// TIA Portal project "IPC200_V15" (V15)

(* hardware
DEVICE "Estación SIMATIC 1200_1"  S71200.Device
   slot 0: "Rack S7-1200"  Rack  V1.0
   slot 1: "IPC201C"  CPU 1214C DC/DC/DC  6ES7 214-1AG40-0XB0  V4.0
   slot 2: "DI8 x 24V DC / DQ8 x relé_1"  6ES7 223-1BH32-0XB0  V2.0
   slot 3: "AI4 x 13bits_1"  6ES7 231-4HD32-0XB0  V2.0
   slot 4: "AQ4 x 14 bits_1"  6ES7 232-4HD32-0XB0  V2.0
DEVICE "S7-1200 station_1"  S7-1200 Station
   slot 0: "Rack_0"  Rack  V1.0
   slot 1: "IPC202B"  CPU 1214C DC/DC/DC  6ES7 214-1AG40-0XB0  V4.0
   slot 2: "DI 16x24VDC_1"  6ES7 221-1BH32-0XB0  V2.0
   slot 3: "DQ 8x24VDC _1"  6ES7 222-1BF32-0XB0  V2.0
DEVICE "S7-1200 station_2"  S7-1200 Station
   slot 0: "Rack_0"  S7-1200 Rack  Rack  V1.0
   slot 1: "PLC_1"  CPU 1214C DC/DC/DC  6ES7 214-1AG40-0XB0  V4.2
   slot 2: "DI 8/DQ 8x24VDC_1"  6ES7 223-1BH32-0XB0  V2.0
   slot 3: "AI 4x13BIT_1"  6ES7 231-4HD32-0XB0  V2.0
   slot 4: "AI 4x13BIT_2"  6ES7 231-4HD32-0XB0  V2.0
*)

// ===== PLC "IPC201C"  CPU 1214C DC/DC/DC =====

VAR_GLOBAL   // PLC tag table "Tabla de variables estándar"
   "A4+" AT %Q0.0 : Bool;   // Auxiliar tank output valve
   "A1+" AT %Q0.1 : Bool;   // Left tank output valve
   "B1+" AT %Q0.2 : Bool;   // Left tank input valve
   "A2+" AT %Q0.3 : Bool;   // Central tank output valve
   "B2+" AT %Q0.4 : Bool;   // Central tank input valve
   "P3+" AT %Q0.5 : Bool;   // Right tank pressure input valve
   "B3+" AT %Q0.6 : Bool;   // Right tank input valve
   "BR" AT %Q0.7 : Bool;   // Red light
   "Invert_VBus" AT %Q1.0 : Bool;   // Switch polarity Peltier cells and run fan
   "plc_reg" AT %Q1.1 : Bool;   // Switch analogue inputs to PLC
   "plc_reg0" AT %Q2.0 : Bool;   // Proportional valve control value from PLC
   "start" AT %I0.0 : Bool;   // Start pushbutton
   "stop" AT %I0.1 : Bool;   // Stop pushbutton
   "I_II" AT %I0.2 : Bool;   // Regulator/PLC
   "reset" AT %I0.3 : Bool;   // Reset pushbutton
   "max1" AT %I0.4 : Bool;   // Maximum left tank level
   "min1" AT %I0.5 : Bool;   // Minimum left tank level
   "max2" AT %I0.6 : Bool;   // Maximum central tank level
   "min2" AT %I0.7 : Bool;   // Minimum central tank level
   "max3" AT %I1.0 : Bool;   // Maximum right tank level
   "min3" AT %I1.1 : Bool;   // Minimum right tank level
   "ps3_out1" AT %I1.2 : Bool;   // Right tank pressure output 1
   "ps3_out2" AT %I1.3 : Bool;   // Right tank pressure output 2
   "dis1_out1" AT %I1.4 : Bool;   // Central tank level output 1
   "dis1_out2" AT %I1.5 : Bool;   // Central tank level output 2
   "dis2_out1" AT %I2.0 : Bool;   // Flow output 1
   "dis2_out2" AT %I2.1 : Bool;   // Flow output 2
   "AnOut1_ITV" AT %MW10 : Int;
   "AnOut2_PV" AT %MW12 : Int;
   "AnOut3_CP" AT %MW14 : Int;
   "AnOut4_PUMP" AT %MW16 : Int;
   "VP_Temp" AT %MW30 : Int;
   "VP_Flow" AT %MW32 : Int;
   "VP_Level" AT %MW34 : Int;
   "VP_P1" AT %MW36 : Int;
   "PID_in_SP" AT %MW88 : Int;
   "PID_out_CS" AT %MW90 : Int;
   "VP_Temp_real" AT %MD40 : Real;
   "VP_Flow_real" AT %MD44 : Real;
   "VP_Level_real" AT %MD48 : Real;
   "VP_Pressure_DEP1_real" AT %MD52 : Real;
   "VP_Pressure_DEP3_real" AT %MD56 : Real;
   "PID_out_CS_real" AT %MD76 : Real;
   "PID_out_Error_real" AT %MD80 : Real;
   "PID_in_SP_real" AT %MD84 : Real;
   "PID_in_PV_real" AT %MD92 : Real;
   "PID_EN" AT %M1.0 : Bool;
   "TK1_MIN" AT %M1.1 : Bool;   // Minimum level reached in DEP1
   "TK2_MIN" AT %M1.2 : Bool;   // Minimum level reached in DEP2
   "TK3_MIN" AT %M1.3 : Bool;   // Minimum level reached in DEP3
   "Running" AT %M1.4 : Bool;   // Station running
   "Set_P" AT %M1.5 : Bool;
   "Set_I" AT %M1.6 : Bool;
   "Set_D" AT %M1.7 : Bool;
   "Run_PID" AT %M2.0 : Bool;   // Activation instruction of PID
   "ITV_out" AT %QW144 : Word;   // Analogue output of ITV
   "P3_out" AT %QW146 : Word;   // Analogue output of proportional valve
   "CP_out" AT %QW148 : Word;   // Analogue output of Peltier cells
   "PUMP_out" AT %QW150 : Word;   // Analogue output of pump
   "FLOW_in" AT %IW114 : Word;   // Value of flow
   "LEVEL_in" AT %IW116 : Word;   // Value of level
   "ITV_in" AT %IW64 : Word;   // Value of pressure in left tank (ITV)
   "P3_in" AT %IW118 : Word;   // Value of pressure in right tank
   "VP_P3" AT %MW38 : Int;
   "TEMP_in" AT %IW112 : Word;   // Value of temperature
   "All_off" AT %M2.7 : Bool;
   "Step_0" AT %M3.0 : Bool;   // Step_0 - Waiting for the station 2 signal
   "Step_1" AT %M3.1 : Bool;   // Step_1 - Start to fill the can
   "Step_2" AT %M3.2 : Bool;   // Step_2 - Stop to fill the can
   "Peltier_V_scada" AT %M20.0 : Bool;   // PC-->PLC
   "Motor_scada" AT %M20.5 : Bool;   // PC-->PLC
   "Fan_scada" AT %M20.6 : Bool;   // PC-->PLC
   "A1+_scada" AT %M21.0 : Bool;   // PC-->PLC
   "B1+_scada" AT %M21.1 : Bool;   // PC-->PLC
   "A2+_scada" AT %M21.2 : Bool;   // PC-->PLC
   "B2+_scada" AT %M21.3 : Bool;   // PC-->PLC
   "P3+_scada" AT %M21.4 : Bool;   // PC-->PLC
   "B3+_scada" AT %M21.5 : Bool;   // PC-->PLC
   "A4+_scada" AT %M21.6 : Bool;   // PC-->PLC
   "A5+_scada" AT %M21.7 : Bool;   // PC-->PLC
   "P_Temp1" AT %M23.0 : Bool;   // PC-->PLC
   "PID_Reverse" AT %M23.1 : Bool;   // PC-->PLC // Reversal of working mode for the cooling action
   "P_Level1" AT %M23.2 : Bool;   // PC-->PLC
   "P_Level2" AT %M23.3 : Bool;   // PC-->PLC
   "P_Level3" AT %M23.4 : Bool;   // PC-->PLC
   "P_Flow1" AT %M23.5 : Bool;   // PC-->PLC
   "P_Flow2" AT %M23.6 : Bool;   // PC-->PLC
   "P_Flow3" AT %M23.7 : Bool;   // PC-->PLC
   "B1+_show_scada" AT %M24.0 : Bool;   // PLC-->PC
   "A2+_show_scada" AT %M24.1 : Bool;   // PLC-->PC
   "B2+_show_scada" AT %M24.2 : Bool;   // PLC-->PC
   "P3+_show_scada" AT %M24.3 : Bool;   // PLC-->PC
   "B3+_show_scada" AT %M24.4 : Bool;   // PLC-->PC
   "A4+_show_scada" AT %M24.5 : Bool;   // PLC-->PC
   "A5+_show_scada" AT %M24.6 : Bool;   // PLC-->PC
   "Min1_scada" AT %M25.0 : Bool;   // PLC-->PC
   "Min2_scada" AT %M25.1 : Bool;   // PLC-->PC
   "Min3_scada" AT %M25.2 : Bool;   // PLC-->PC
   "Max1_scada" AT %M25.3 : Bool;   // PLC-->PC
   "Max2_scada" AT %M25.4 : Bool;   // PLC-->PC
   "Max3_scada" AT %M25.5 : Bool;   // PLC-->PC
   "I_II_scada" AT %M25.6 : Bool;   // PLC-->PC
   "A1+_show_scada" AT %M25.7 : Bool;   // PLC-->PC
   "start_scada" AT %M29.6 : Bool;   // Start from the SCADA
   "stop_scada" AT %M29.7 : Bool;   // Stop from the SCADA
   "Tag_11" AT %MW20 : Word;
   "Clock_Byte" AT %MB0 : Byte;
   "Clock_10Hz" AT %M0.0 : Bool;
   "Clock_5Hz" AT %M0.1 : Bool;
   "Clock_2.5Hz" AT %M0.2 : Bool;
   "Clock_2Hz" AT %M0.3 : Bool;
   "Clock_1.25Hz" AT %M0.4 : Bool;
   "Clock_1Hz" AT %M0.5 : Bool;
   "Clock_0.625Hz" AT %M0.6 : Bool;
   "Clock_0.5Hz" AT %M0.7 : Bool;
   "P_Gain_scada_real" AT %MD60 : Real;
   "I_Time_scada_real" AT %MD64 : Real;
   "D_Time_scada_real" AT %MD68 : Real;
   "plc_reg1" AT %Q2.1 : Bool;   // ITV SetPoint from PLC
   "event_flow" AT %Q2.2 : Bool;   // Stop industrial flow controller
   "Temp1_E5CNH" AT %M22.0 : Bool;   // PC-->PLC
   "Level_aux1" AT %MD72 : UDInt;
   "Level_aux2" AT %MD96 : UDInt;
   "Level_aux3" AT %MW100 : Int;
   "Tag_10" AT %MW22 : Word;
   "Temp2_E5CNH" AT %M22.1 : Bool;   // PC-->PLC
   "Tag_13" AT %M589.0 : Bool;
   "P_Gain" AT %MD102 : Real;
   "I_Time" AT %MD106 : Real;
   "D_Time" AT %MD110 : Real;
   "P_Gain_scada" AT %MD114 : DWord;
   "I_Time_scada" AT %MD118 : DWord;
   "D_Time_scada" AT %MD122 : DWord;
   "Tag_14" AT %M400.0 : Bool;
   "Tag_15" AT %M589.1 : Bool;
   "Tag_16" AT %M589.2 : Bool;
   "VP_Temp_aux" AT %MW126 : Int;
   "PID_in_SP_aux" AT %MW128 : Int;
   "event_level" AT %Q2.3 : Bool;   // Stop industrial level controller
   "plc_reg2" AT %Q2.4 : Bool;   // Switch between flow and level control
   "A5+" AT %Q2.5 : Bool;   // Pump run
   "PLC_reg_sensor_scada" AT %M20.1 : Bool;   // PC-->PLC
   "PLC_reg0_scada" AT %M20.2 : Bool;   // PC-->PLC
   "PLC_reg1_scada" AT %M20.3 : Bool;   // PC-->PLC
   "PLC_reg2_scada" AT %M20.4 : Bool;   // PC-->PLC
   "Level1_E5CNH" AT %M22.2 : Bool;   // PC-->PLC
   "Level2_E5CNH" AT %M22.3 : Bool;   // PC-->PLC
   "Level3_E5CNH" AT %M22.4 : Bool;   // PC-->PLC
   "Flow1_E5CNH" AT %M22.5 : Bool;   // PC-->PLC
   "Flow2_E5CNH" AT %M22.6 : Bool;   // PC-->PLC
   "Flow3_E5CNH" AT %M22.7 : Bool;   // PC-->PLC
   "IPC2_on" AT %I10.0 : Bool;   // IPC202 active
   "IPC1_StartCycle" AT %I10.1 : Bool;   // Start cycle in IPC201C from IPC202
   "IPC1_on" AT %Q10.0 : Bool;   // IPC201C active to IPC202
   "IPC1_end" AT %Q10.1 : Bool;   // End cycle of IPC201C to IPC202
   "IPC1_full" AT %Q10.2 : Bool;   // Central tank full in IPC201C to IPC202
   "Tag_1" AT %IB10 : Byte;
   "TEMP_PRG" AT %M11.0 : Bool;   // Temporary parameter
   "PRG_FLAG" AT %M11.3 : Bool;   // Program is running
   "KORAK" AT %MW110 : UInt;
END_VAR

DATA_BLOCK "apple_juice_program_DB"   // DB45
{ S7_Optimized_Access := 'TRUE' }
VERSION : 0.1
// stored: InstanceOfName APPLE_JUICE_PROCESS
"APPLE_JUICE_PROCESS"
BEGIN
END_DATA_BLOCK

// folder: System blocks/Program resources

DATA_BLOCK "TIMER_1"   // DB5
{ S7_Optimized_Access := 'TRUE' }
AUTHOR : Simatic
FAMILY : IEC
NAME : IEC_TMR
VERSION : 1.0
// stored: InstanceOfName IEC_TIMER
"IEC_TIMER"
BEGIN
END_DATA_BLOCK

DATA_BLOCK "TIMER_2"   // DB6
{ S7_Optimized_Access := 'TRUE' }
AUTHOR : Simatic
FAMILY : IEC
NAME : IEC_TMR
VERSION : 1.0
// stored: InstanceOfName IEC_TIMER
"IEC_TIMER"
BEGIN
END_DATA_BLOCK

DATA_BLOCK "TIMER_3"   // DB7
{ S7_Optimized_Access := 'TRUE' }
AUTHOR : Simatic
FAMILY : IEC
NAME : IEC_TMR
VERSION : 1.0
// stored: InstanceOfName IEC_TIMER
"IEC_TIMER"
BEGIN
END_DATA_BLOCK

DATA_BLOCK "TIMER_4"   // DB8
{ S7_Optimized_Access := 'TRUE' }
AUTHOR : Simatic
FAMILY : IEC
NAME : IEC_TMR
VERSION : 1.0
// stored: InstanceOfName IEC_TIMER
"IEC_TIMER"
BEGIN
END_DATA_BLOCK

DATA_BLOCK "TIMER_5"   // DB9
{ S7_Optimized_Access := 'TRUE' }
AUTHOR : Simatic
FAMILY : IEC
NAME : IEC_TMR
VERSION : 1.0
// stored: InstanceOfName IEC_TIMER
"IEC_TIMER"
BEGIN
END_DATA_BLOCK

DATA_BLOCK "TIMER_6"   // DB10
{ S7_Optimized_Access := 'TRUE' }
AUTHOR : Simatic
FAMILY : IEC
NAME : IEC_TMR
VERSION : 1.0
// stored: InstanceOfName IEC_TIMER
"IEC_TIMER"
BEGIN
END_DATA_BLOCK

DATA_BLOCK "TIMER_7"   // DB11
{ S7_Optimized_Access := 'TRUE' }
AUTHOR : Simatic
FAMILY : IEC
NAME : IEC_TMR
VERSION : 1.0
// stored: InstanceOfName IEC_TIMER
"IEC_TIMER"
BEGIN
END_DATA_BLOCK

DATA_BLOCK "TIMER_8"   // DB12
{ S7_Optimized_Access := 'TRUE' }
AUTHOR : Simatic
FAMILY : IEC
NAME : IEC_TMR
VERSION : 1.0
// stored: InstanceOfName IEC_TIMER
"IEC_TIMER"
BEGIN
END_DATA_BLOCK

DATA_BLOCK "TIMER_9"   // DB13
{ S7_Optimized_Access := 'TRUE' }
AUTHOR : Simatic
FAMILY : IEC
NAME : IEC_TMR
VERSION : 1.0
// stored: InstanceOfName IEC_TIMER
"IEC_TIMER"
BEGIN
END_DATA_BLOCK

DATA_BLOCK "TIMER_PROG_2"   // DB17
{ S7_Optimized_Access := 'TRUE' }
AUTHOR : Simatic
FAMILY : IEC
NAME : IEC_TMR
VERSION : 1.0
// stored: InstanceOfName IEC_TIMER
"IEC_TIMER"
BEGIN
END_DATA_BLOCK

DATA_BLOCK "TIMER_PROG_1"   // DB19
{ S7_Optimized_Access := 'TRUE' }
AUTHOR : Simatic
FAMILY : IEC
NAME : IEC_TMR
VERSION : 1.0
// stored: InstanceOfName IEC_TIMER
"IEC_TIMER"
BEGIN
END_DATA_BLOCK

DATA_BLOCK "TIMER_PROG_3"   // DB20
{ S7_Optimized_Access := 'TRUE' }
AUTHOR : Simatic
FAMILY : IEC
NAME : IEC_TMR
VERSION : 1.0
// stored: InstanceOfName IEC_TIMER
"IEC_TIMER"
BEGIN
END_DATA_BLOCK

DATA_BLOCK "TIMER_PROG_4"   // DB21
{ S7_Optimized_Access := 'TRUE' }
AUTHOR : Simatic
FAMILY : IEC
NAME : IEC_TMR
VERSION : 1.0
// stored: InstanceOfName IEC_TIMER
"IEC_TIMER"
BEGIN
END_DATA_BLOCK

DATA_BLOCK "TIMER_PROG_5"   // DB22
{ S7_Optimized_Access := 'TRUE' }
AUTHOR : Simatic
FAMILY : IEC
NAME : IEC_TMR
VERSION : 1.0
// stored: InstanceOfName IEC_TIMER
"IEC_TIMER"
BEGIN
END_DATA_BLOCK

DATA_BLOCK "TIMER_PROG_6"   // DB23
{ S7_Optimized_Access := 'TRUE' }
AUTHOR : Simatic
FAMILY : IEC
NAME : IEC_TMR
VERSION : 1.0
// stored: InstanceOfName IEC_TIMER
"IEC_TIMER"
BEGIN
END_DATA_BLOCK

DATA_BLOCK "TIMER_PROG_7"   // DB24
{ S7_Optimized_Access := 'TRUE' }
AUTHOR : Simatic
FAMILY : IEC
NAME : IEC_TMR
VERSION : 1.0
// stored: InstanceOfName IEC_TIMER
"IEC_TIMER"
BEGIN
END_DATA_BLOCK

DATA_BLOCK "TIMER_PROG_8"   // DB25
{ S7_Optimized_Access := 'TRUE' }
AUTHOR : Simatic
FAMILY : IEC
NAME : IEC_TMR
VERSION : 1.0
// stored: InstanceOfName IEC_TIMER
"IEC_TIMER"
BEGIN
END_DATA_BLOCK

DATA_BLOCK "TIMER_PROG_9"   // DB26
{ S7_Optimized_Access := 'TRUE' }
AUTHOR : Simatic
FAMILY : IEC
NAME : IEC_TMR
VERSION : 1.0
// stored: InstanceOfName IEC_TIMER
"IEC_TIMER"
BEGIN
END_DATA_BLOCK

DATA_BLOCK "TIMER_PROG_10"   // DB27
{ S7_Optimized_Access := 'TRUE' }
AUTHOR : Simatic
FAMILY : IEC
NAME : IEC_TMR
VERSION : 1.0
// stored: InstanceOfName IEC_TIMER
"IEC_TIMER"
BEGIN
END_DATA_BLOCK

DATA_BLOCK "TIMER_PROG_24"   // DB28
{ S7_Optimized_Access := 'TRUE' }
AUTHOR : Simatic
FAMILY : IEC
NAME : IEC_TMR
VERSION : 1.0
// stored: InstanceOfName IEC_TIMER
"IEC_TIMER"
BEGIN
END_DATA_BLOCK

DATA_BLOCK "TIMER_PROG_12"   // DB29
{ S7_Optimized_Access := 'TRUE' }
AUTHOR : Simatic
FAMILY : IEC
NAME : IEC_TMR
VERSION : 1.0
// stored: InstanceOfName IEC_TIMER
"IEC_TIMER"
BEGIN
END_DATA_BLOCK

DATA_BLOCK "IEC_Counter_0_DB"   // DB30
{ S7_Optimized_Access := 'TRUE' }
AUTHOR : Simatic
FAMILY : IEC
NAME : CNTR
VERSION : 1.0
// stored: InstanceOfName IEC_COUNTER
"IEC_COUNTER"
BEGIN
END_DATA_BLOCK

DATA_BLOCK "TIMER_PROG_13"   // DB31
{ S7_Optimized_Access := 'TRUE' }
AUTHOR : Simatic
FAMILY : IEC
NAME : IEC_TMR
VERSION : 1.0
// stored: InstanceOfName IEC_TIMER
"IEC_TIMER"
BEGIN
END_DATA_BLOCK

DATA_BLOCK "IEC_Counter_0_DB_1"   // DB32
{ S7_Optimized_Access := 'TRUE' }
AUTHOR : Simatic
FAMILY : IEC
NAME : CNTR
VERSION : 1.0
// stored: InstanceOfName IEC_COUNTER
"IEC_COUNTER"
BEGIN
END_DATA_BLOCK

DATA_BLOCK "TIMER_PROG_14"   // DB33
{ S7_Optimized_Access := 'TRUE' }
AUTHOR : Simatic
FAMILY : IEC
NAME : IEC_TMR
VERSION : 1.0
// stored: InstanceOfName IEC_TIMER
"IEC_TIMER"
BEGIN
END_DATA_BLOCK

DATA_BLOCK "TIMER_PROG_15"   // DB34
{ S7_Optimized_Access := 'TRUE' }
AUTHOR : Simatic
FAMILY : IEC
NAME : IEC_TMR
VERSION : 1.0
// stored: InstanceOfName IEC_TIMER
"IEC_TIMER"
BEGIN
END_DATA_BLOCK

DATA_BLOCK "TIMER_PROG_16"   // DB35
{ S7_Optimized_Access := 'TRUE' }
AUTHOR : Simatic
FAMILY : IEC
NAME : IEC_TMR
VERSION : 1.0
// stored: InstanceOfName IEC_TIMER
"IEC_TIMER"
BEGIN
END_DATA_BLOCK

DATA_BLOCK "TIMER_PROG_17"   // DB36
{ S7_Optimized_Access := 'TRUE' }
AUTHOR : Simatic
FAMILY : IEC
NAME : IEC_TMR
VERSION : 1.0
// stored: InstanceOfName IEC_TIMER
"IEC_TIMER"
BEGIN
END_DATA_BLOCK

DATA_BLOCK "TIMER_PROG_18"   // DB37
{ S7_Optimized_Access := 'TRUE' }
AUTHOR : Simatic
FAMILY : IEC
NAME : IEC_TMR
VERSION : 1.0
// stored: InstanceOfName IEC_TIMER
"IEC_TIMER"
BEGIN
END_DATA_BLOCK

DATA_BLOCK "IEC_Counter_0_DB_2"   // DB38
{ S7_Optimized_Access := 'TRUE' }
AUTHOR : Simatic
FAMILY : IEC
NAME : CNTR
VERSION : 1.0
// stored: InstanceOfName IEC_COUNTER
"IEC_COUNTER"
BEGIN
END_DATA_BLOCK

DATA_BLOCK "TIMER_PROG_19"   // DB39
{ S7_Optimized_Access := 'TRUE' }
AUTHOR : Simatic
FAMILY : IEC
NAME : IEC_TMR
VERSION : 1.0
// stored: InstanceOfName IEC_TIMER
"IEC_TIMER"
BEGIN
END_DATA_BLOCK

DATA_BLOCK "TIMER_PROG_20"   // DB40
{ S7_Optimized_Access := 'TRUE' }
AUTHOR : Simatic
FAMILY : IEC
NAME : IEC_TMR
VERSION : 1.0
// stored: InstanceOfName IEC_TIMER
"IEC_TIMER"
BEGIN
END_DATA_BLOCK

DATA_BLOCK "TIMER_PROG_21"   // DB41
{ S7_Optimized_Access := 'TRUE' }
AUTHOR : Simatic
FAMILY : IEC
NAME : IEC_TMR
VERSION : 1.0
// stored: InstanceOfName IEC_TIMER
"IEC_TIMER"
BEGIN
END_DATA_BLOCK

DATA_BLOCK "TIMER_PROG_22"   // DB42
{ S7_Optimized_Access := 'TRUE' }
AUTHOR : Simatic
FAMILY : IEC
NAME : IEC_TMR
VERSION : 1.0
// stored: InstanceOfName IEC_TIMER
"IEC_TIMER"
BEGIN
END_DATA_BLOCK

DATA_BLOCK "TIMER_PROG_23"   // DB43
{ S7_Optimized_Access := 'TRUE' }
AUTHOR : Simatic
FAMILY : IEC
NAME : IEC_TMR
VERSION : 1.0
// stored: InstanceOfName IEC_TIMER
"IEC_TIMER"
BEGIN
END_DATA_BLOCK

DATA_BLOCK "IEC_Counter_0_DB_3"   // DB44
{ S7_Optimized_Access := 'TRUE' }
AUTHOR : Simatic
FAMILY : IEC
NAME : CNTR
VERSION : 1.0
// stored: InstanceOfName IEC_COUNTER
"IEC_COUNTER"
BEGIN
END_DATA_BLOCK

DATA_BLOCK "IEC_Timer_0_DB_1"   // DB52
{ S7_Optimized_Access := 'TRUE' }
AUTHOR : Simatic
FAMILY : IEC
NAME : IEC_TMR
VERSION : 1.0
// stored: InstanceOfName IEC_TIMER
"IEC_TIMER"
BEGIN
END_DATA_BLOCK

DATA_BLOCK "IEC_Timer_0_DB"   // DB53
{ S7_Optimized_Access := 'TRUE' }
AUTHOR : Simatic
FAMILY : IEC
NAME : IEC_TMR
VERSION : 1.0
// stored: InstanceOfName IEC_TIMER
"IEC_TIMER"
BEGIN
END_DATA_BLOCK

// folder: (top level)

FUNCTION_BLOCK "APPLE_JUICE_PROCESS"   // FB1, SCL
{ S7_Optimized_Access := 'TRUE' }
VERSION : 0.1
   VAR
      currentState : Int := 0;
      "timer" : Time;
      onDelayCheck : Bool;
      fallingEgdeDedect1 : Bool;
      fallingEgdeDedect : Bool;
      risingEgdeDedect : Bool;
      processFinished : Bool;
   END_VAR
   VAR CONSTANT
      STATE_WAIT_FOR_START : Int := -1;
      STATE_START_FILL_WATER : Int;
      STATE_WAIT_FOR_FILL_WATER_TANK : Int := 1;
      FILL_WAIT : Time := T#5s;
      STATE_START_FILL_APPLE : Int := 2;
      STATE_WAIT_FILL_APPLE : Int := 3;
      STATE_START_FILL_APPLE_JUICE_WITH_WATER : Int := 4;
      STATE_WAIT_FILL_APPLE_JUICE_WITH_WATER : Int := 5;
      STATE_START_FILL_APPLE_JUICE_WITH_APPLE : Int := 6;
      STATE_WAIT_FILL_APPLE_JUICE_WITH_APPLE : Int := 7;
      STATE_START_FILL_OUT_APPLE : Int := 8;
      STATE_WAIT_FILL_OUT_APPLE : Int := 9;
      STATE_WAIT_FOR_NEXT_PROCESS : Int := 10;
      PUMP_CHARGE : Int := 8000;
      VALVE_CHARE : Int := 20000;
   END_VAR
BEGIN
   CASE #currentState OF
       #STATE_WAIT_FOR_START:
           "R_TRIG_DB_1"(CLK:="start",
                         Q=>#risingEgdeDedect);

           IF #risingEgdeDedect = TRUE THEN
               #currentState := #STATE_START_FILL_WATER;
           END_IF;

       #STATE_START_FILL_WATER:
           "START_LOAD_TANK"(feedback1 := "A4+",
                             feedback2 := "A5+",
                             feedback3 := "B1+",
                             command1 => "A4+_scada",
                             command2 => "A5+_scada",
                             command3 => "B1+_scada",
                             pumpValue := #PUMP_CHARGE,
                             pumpOutput => "AnOut4_PUMP",
                             routeReady => #processFinished);

           IF #processFinished = TRUE THEN
               #currentState := #STATE_WAIT_FOR_FILL_WATER_TANK;
           END_IF;

       #STATE_WAIT_FOR_FILL_WATER_TANK:
           "F_TRIG_DB"(CLK := "max1",
                       Q => #fallingEgdeDedect);

           IF #fallingEgdeDedect = TRUE OR "max1" = FALSE THEN
               "STOP_LOAD_TANK"(command1 => "A4+_scada",
                                command2 => "A5+_scada",
                                command3 => "B1+_scada",
                                pumpOutput => "AnOut4_PUMP");

               #currentState := #STATE_START_FILL_APPLE;
           END_IF;

       #STATE_START_FILL_APPLE:
           "START_LOAD_TANK"(feedback1 := "A4+",
                             feedback2 := "A5+",
                             feedback3 := "B3+",
                             command1 => "A4+_scada",
                             command2 => "A5+_scada",
                             command3 => "B3+_scada",
                             pumpValue := #PUMP_CHARGE,
                             pumpOutput => "AnOut4_PUMP",
                             routeReady => #processFinished);

           IF #processFinished = TRUE THEN
               #currentState := #STATE_WAIT_FILL_APPLE;
           END_IF;

       #STATE_WAIT_FILL_APPLE:
           "F_TRIG_DB_1"(CLK := "max3",
                         Q => #fallingEgdeDedect);

           IF #fallingEgdeDedect = TRUE OR "max3" = FALSE THEN
               "STOP_LOAD_TANK"(command1 => "A4+_scada",
                                command2 => "A5+_scada",
                                command3 => "B3+_scada",
                                pumpOutput => "AnOut4_PUMP");

               #currentState := #STATE_START_FILL_APPLE_JUICE_WITH_WATER;
           END_IF;

       #STATE_START_FILL_APPLE_JUICE_WITH_WATER:
           "START_LOAD_APPLE_JUICE_TANK"(feedback1 := "A1+",
                                         feedback2 := "B2+",
                                         command1 => "A1+_scada",
                                         command2 => "B2+_scada",
                                         regulatorCommand => "PLC_reg1_scada",
                                         analogValue := #VALVE_CHARE,
                                         analogOutput => "AnOut1_ITV",
                                         routeReady => #processFinished);

           IF #processFinished = TRUE THEN
               #currentState := #STATE_WAIT_FILL_APPLE_JUICE_WITH_WATER;
           END_IF;

       #STATE_WAIT_FILL_APPLE_JUICE_WITH_WATER:
           "R_TRIG_DB"(CLK := "min2",
                       Q => #risingEgdeDedect);

           IF #risingEgdeDedect = TRUE OR "min2" = TRUE THEN
               "STOP_LOAD_APPLE_JUICE_TANK"(command1 => "A1+_scada",
                                            command2 => "B2+_scada",
                                            regulatorCommand => "PLC_reg0_scada",
                                            analogOutput => "AnOut1_ITV");

               #currentState := #STATE_START_FILL_APPLE_JUICE_WITH_APPLE;
           END_IF;

       #STATE_START_FILL_APPLE_JUICE_WITH_APPLE:
           "START_LOAD_APPLE_JUICE_TANK"(feedback1 := "P3+",
                                         feedback2 := "B2+",
                                         command1 => "P3+_scada",
                                         command2 => "B2+_scada",
                                         regulatorCommand => "PLC_reg0_scada",
                                         analogValue := #VALVE_CHARE,
                                         analogOutput => "AnOut2_PV",
                                         routeReady => #processFinished);

           IF #processFinished = TRUE THEN
               #currentState := #STATE_WAIT_FILL_APPLE_JUICE_WITH_APPLE;
           END_IF;

       #STATE_WAIT_FILL_APPLE_JUICE_WITH_APPLE:
           "F_TRIG_DB_2"(CLK := "min3",
                         Q => #fallingEgdeDedect);
           "F_TRIG_DB_3"(CLK := "max2",
                         Q => #fallingEgdeDedect1);



           IF (#fallingEgdeDedect = TRUE OR "min3" = FALSE) OR
               (#fallingEgdeDedect1 = TRUE OR "max2" = FALSE) THEN
               "STOP_LOAD_APPLE_JUICE_TANK"(command1 => "P3+_scada",
                                            command2 => "B2+_scada",
                                            regulatorCommand => "PLC_reg1_scada",
                                            analogOutput => "AnOut2_PV");

               #currentState := #STATE_START_FILL_OUT_APPLE;
           END_IF;

       #STATE_START_FILL_OUT_APPLE:
           "FILL_APPLE_TO_BOTTLE"(feedback1 := "A2+",
                                  feedback2 := "A5+",
                                  command1 => "A2+_scada",
                                  command2 => "A5+_scada",
                                  analogValue := 8000,
                                  analogOutput => "AnOut4_PUMP",
                                  routeReady => #processFinished);

           IF #processFinished = TRUE THEN
               #currentState := #STATE_WAIT_FILL_OUT_APPLE;
           END_IF;

       #STATE_WAIT_FILL_OUT_APPLE:
           "IEC_Timer_0_DB".TON(IN := TRUE,
                                PT := T#40s,
                                Q => #onDelayCheck,
                                ET => #timer);


           IF #onDelayCheck = TRUE THEN
               "STOP_FILL_APPLE_TO_BOTTLE"(command1 => "A2+_scada",
                                           command2 => "A5+_scada",
                                           analogOutput => "AnOut4_PUMP");

               "IEC_Timer_0_DB".TON(IN := FALSE,
                                    PT := T#40s,
                                    Q => #onDelayCheck,
                                    ET => #timer);

               #currentState := #STATE_WAIT_FOR_START;
           END_IF;
   END_CASE;
END_FUNCTION_BLOCK

FUNCTION "TIMERS" : Void   // FC1, LAD
TITLE = TIMERS
{ S7_Optimized_Access := 'TRUE' }
VERSION : 0.1
BEGIN

REGION Network 1: TIMER 1
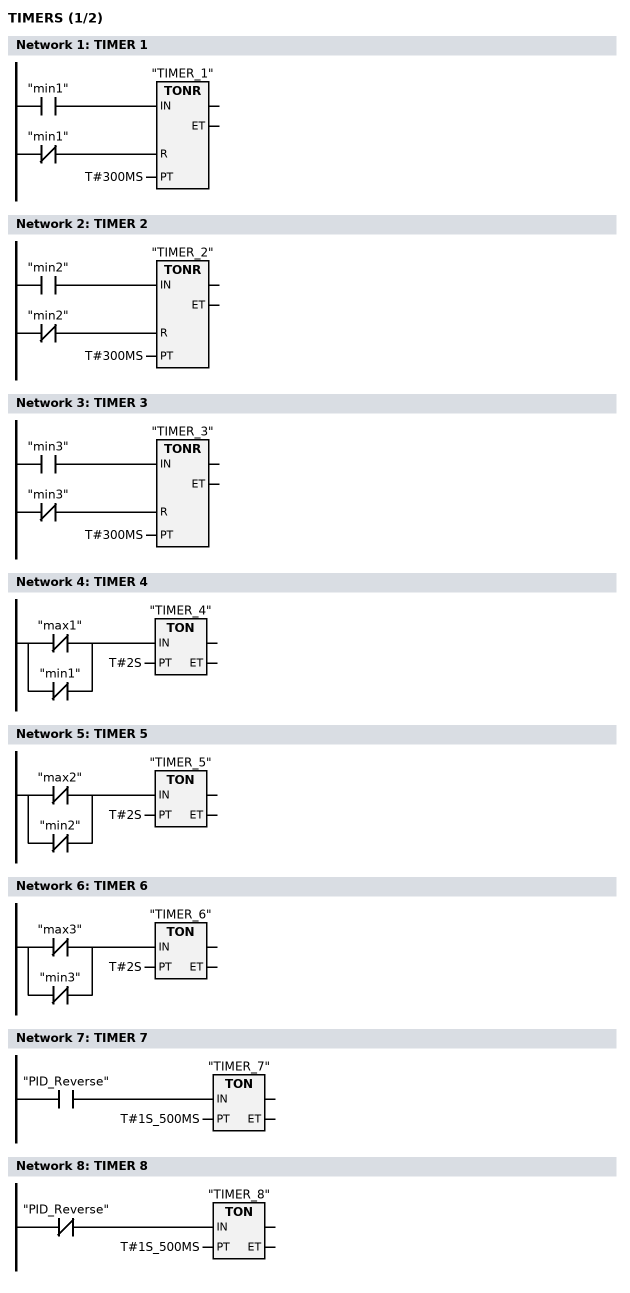
   "TIMER_1".TONR(IN := "min1", R := NOT "min1", PT := T#300MS);
END_REGION

REGION Network 2: TIMER 2
   "TIMER_2".TONR(IN := "min2", R := NOT "min2", PT := T#300MS);
END_REGION

REGION Network 3: TIMER 3
   "TIMER_3".TONR(IN := "min3", R := NOT "min3", PT := T#300MS);
END_REGION

REGION Network 4: TIMER 4
   "TIMER_4".TON(IN := NOT "max1" OR NOT "min1", PT := T#2S);
END_REGION

REGION Network 5: TIMER 5
   "TIMER_5".TON(IN := NOT "max2" OR NOT "min2", PT := T#2S);
END_REGION

REGION Network 6: TIMER 6
   "TIMER_6".TON(IN := NOT "max3" OR NOT "min3", PT := T#2S);
END_REGION

REGION Network 7: TIMER 7
   "TIMER_7".TON(IN := "PID_Reverse", PT := T#1S_500MS);
END_REGION

REGION Network 8: TIMER 8
   "TIMER_8".TON(IN := NOT "PID_Reverse", PT := T#1S_500MS);
END_REGION

REGION Network 9: TIMER 9
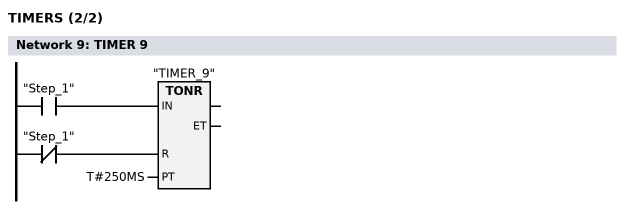
   "TIMER_9".TONR(IN := "Step_1", R := NOT "Step_1", PT := T#250MS);
END_REGION
END_FUNCTION

FUNCTION "WORKBITS" : Void   // FC2, LAD
TITLE = WORKBITS
{ S7_Optimized_Access := 'TRUE' }
VERSION : 0.1
BEGIN

REGION Network 1: TK1_MIN
   // Min level reached in DEP1
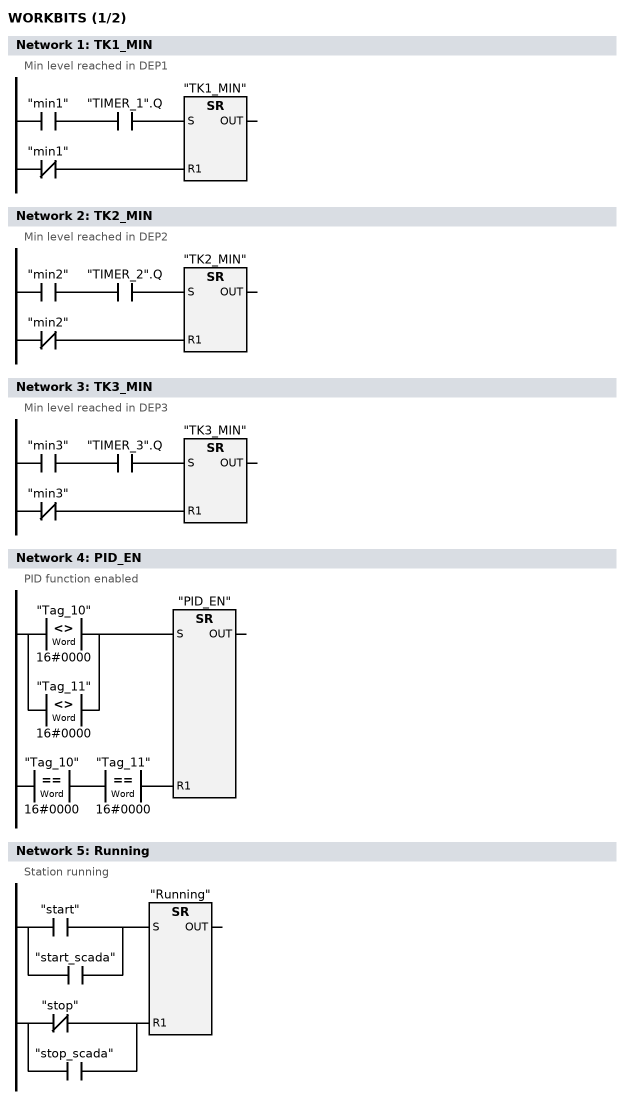
   RUNG wire#powerrail
      Contact( "min1" )
      Contact( "TIMER_1".Q )
      S_SR(operand := "TK1_MIN", r1 := wire#w1)
   END_RUNG
   RUNG wire#powerrail
      I_Contact( "min1" )
   END_RUNG wire#w1
   // the same network as SCL:
   IF "min1" AND "TIMER_1".Q THEN
       "TK1_MIN" := TRUE;   // SR flip-flop
   END_IF;
   IF NOT "min1" THEN "TK1_MIN" := FALSE; END_IF;
END_REGION

REGION Network 2: TK2_MIN
   // Min level reached in DEP2
   RUNG wire#powerrail
      Contact( "min2" )
      Contact( "TIMER_2".Q )
      S_SR(operand := "TK2_MIN", r1 := wire#w1)
   END_RUNG
   RUNG wire#powerrail
      I_Contact( "min2" )
   END_RUNG wire#w1
   // the same network as SCL:
   IF "min2" AND "TIMER_2".Q THEN
       "TK2_MIN" := TRUE;   // SR flip-flop
   END_IF;
   IF NOT "min2" THEN "TK2_MIN" := FALSE; END_IF;
END_REGION

REGION Network 3: TK3_MIN
   // Min level reached in DEP3
   RUNG wire#powerrail
      Contact( "min3" )
      Contact( "TIMER_3".Q )
      S_SR(operand := "TK3_MIN", r1 := wire#w1)
   END_RUNG
   RUNG wire#powerrail
      I_Contact( "min3" )
   END_RUNG wire#w1
   // the same network as SCL:
   IF "min3" AND "TIMER_3".Q THEN
       "TK3_MIN" := TRUE;   // SR flip-flop
   END_IF;
   IF NOT "min3" THEN "TK3_MIN" := FALSE; END_IF;
END_REGION

REGION Network 4: PID_EN
   // PID function enabled
   RUNG wire#powerrail
      { S7_Templates := "SrcType := Word" } NE_Contact(in1 := "Tag_10", in2 := 16#0000)
      wire#w1
      S_SR(operand := "PID_EN", r1 := wire#w2)
   END_RUNG
   RUNG wire#powerrail
      { S7_Templates := "SrcType := Word" } NE_Contact(in1 := "Tag_11", in2 := 16#0000)
   END_RUNG wire#w1
   RUNG wire#powerrail
      { S7_Templates := "SrcType := Word" } EQ_Contact(in1 := "Tag_10", in2 := 16#0000)
      { S7_Templates := "SrcType := Word" } EQ_Contact(in1 := "Tag_11", in2 := 16#0000)
   END_RUNG wire#w2
   // the same network as SCL:
   IF ("Tag_10" <> 16#0000) OR ("Tag_11" <> 16#0000) THEN
       "PID_EN" := TRUE;   // SR flip-flop
   END_IF;
   IF ("Tag_10" = 16#0000) AND ("Tag_11" = 16#0000) THEN "PID_EN" := FALSE; END_IF;
END_REGION

REGION Network 5: Running
   // Station running
   RUNG wire#powerrail
      Contact( "start" )
      wire#w1
      S_SR(operand := "Running", r1 := wire#w2)
   END_RUNG
   RUNG wire#powerrail
      Contact( "start_scada" )
   END_RUNG wire#w1
   RUNG wire#powerrail
      I_Contact( "stop" )
   END_RUNG wire#w2
   RUNG wire#powerrail
      Contact( "stop_scada" )
   END_RUNG wire#w2
   // the same network as SCL:
   IF "start" OR "start_scada" THEN
       "Running" := TRUE;   // SR flip-flop
   END_IF;
   IF NOT "stop" OR "stop_scada" THEN "Running" := FALSE; END_IF;
END_REGION

REGION Network 6: Run_PID
   // Activation instruction of PID
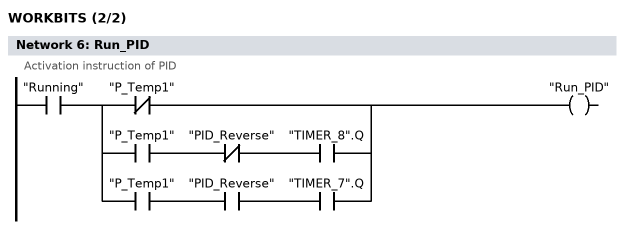
   RUNG wire#powerrail
      Contact( "Running" )
      wire#w1
      I_Contact( "P_Temp1" )
      wire#w2
      Coil( "Run_PID" )
   END_RUNG
   RUNG wire#w1
      Contact( "P_Temp1" )
      I_Contact( "PID_Reverse" )
      Contact( "TIMER_8".Q )
   END_RUNG wire#w2
   RUNG wire#w1
      Contact( "P_Temp1" )
      Contact( "PID_Reverse" )
      Contact( "TIMER_7".Q )
   END_RUNG wire#w2
   // the same network as SCL:
   "Run_PID" := "Running" AND (NOT "P_Temp1" OR ("P_Temp1" AND NOT "PID_Reverse" AND "TIMER_8".Q) OR ("P_Temp1" AND "PID_Reverse" AND "TIMER_7".Q));
END_REGION
END_FUNCTION

FUNCTION "SCADA" : Void   // FC3, LAD
TITLE = Communication between SCADA (PC) and PLC
{ S7_Optimized_Access := 'TRUE' }
VERSION : 0.1
BEGIN

REGION Network 1: PLC-->PLC
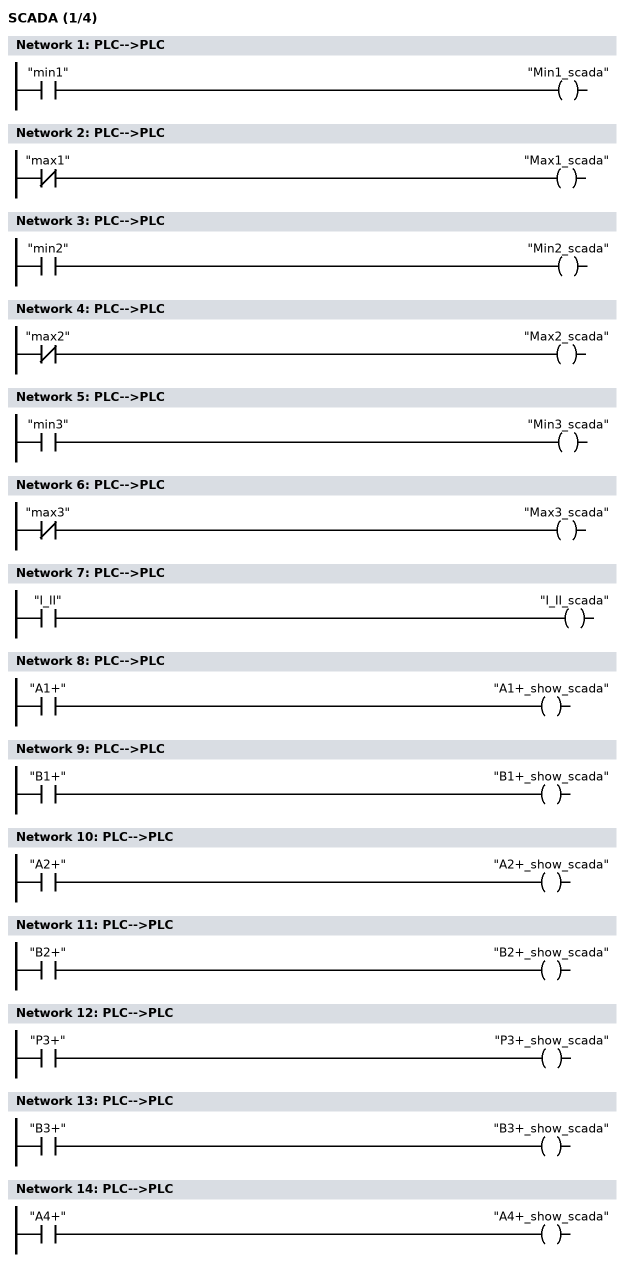
   RUNG wire#powerrail
      Contact( "min1" )
      Coil( "Min1_scada" )
   END_RUNG
   // the same network as SCL:
   "Min1_scada" := "min1";
END_REGION

REGION Network 2: PLC-->PLC
   RUNG wire#powerrail
      I_Contact( "max1" )
      Coil( "Max1_scada" )
   END_RUNG
   // the same network as SCL:
   "Max1_scada" := NOT "max1";
END_REGION

REGION Network 3: PLC-->PLC
   RUNG wire#powerrail
      Contact( "min2" )
      Coil( "Min2_scada" )
   END_RUNG
   // the same network as SCL:
   "Min2_scada" := "min2";
END_REGION

REGION Network 4: PLC-->PLC
   RUNG wire#powerrail
      I_Contact( "max2" )
      Coil( "Max2_scada" )
   END_RUNG
   // the same network as SCL:
   "Max2_scada" := NOT "max2";
END_REGION

REGION Network 5: PLC-->PLC
   RUNG wire#powerrail
      Contact( "min3" )
      Coil( "Min3_scada" )
   END_RUNG
   // the same network as SCL:
   "Min3_scada" := "min3";
END_REGION

REGION Network 6: PLC-->PLC
   RUNG wire#powerrail
      I_Contact( "max3" )
      Coil( "Max3_scada" )
   END_RUNG
   // the same network as SCL:
   "Max3_scada" := NOT "max3";
END_REGION

REGION Network 7: PLC-->PLC
   RUNG wire#powerrail
      Contact( "I_II" )
      Coil( "I_II_scada" )
   END_RUNG
   // the same network as SCL:
   "I_II_scada" := "I_II";
END_REGION

REGION Network 8: PLC-->PLC
   RUNG wire#powerrail
      Contact( "A1+" )
      Coil( "A1+_show_scada" )
   END_RUNG
   // the same network as SCL:
   "A1+_show_scada" := "A1+";
END_REGION

REGION Network 9: PLC-->PLC
   RUNG wire#powerrail
      Contact( "B1+" )
      Coil( "B1+_show_scada" )
   END_RUNG
   // the same network as SCL:
   "B1+_show_scada" := "B1+";
END_REGION

REGION Network 10: PLC-->PLC
   RUNG wire#powerrail
      Contact( "A2+" )
      Coil( "A2+_show_scada" )
   END_RUNG
   // the same network as SCL:
   "A2+_show_scada" := "A2+";
END_REGION

REGION Network 11: PLC-->PLC
   RUNG wire#powerrail
      Contact( "B2+" )
      Coil( "B2+_show_scada" )
   END_RUNG
   // the same network as SCL:
   "B2+_show_scada" := "B2+";
END_REGION

REGION Network 12: PLC-->PLC
   RUNG wire#powerrail
      Contact( "P3+" )
      Coil( "P3+_show_scada" )
   END_RUNG
   // the same network as SCL:
   "P3+_show_scada" := "P3+";
END_REGION

REGION Network 13: PLC-->PLC
   RUNG wire#powerrail
      Contact( "B3+" )
      Coil( "B3+_show_scada" )
   END_RUNG
   // the same network as SCL:
   "B3+_show_scada" := "B3+";
END_REGION

REGION Network 14: PLC-->PLC
   RUNG wire#powerrail
      Contact( "A4+" )
      Coil( "A4+_show_scada" )
   END_RUNG
   // the same network as SCL:
   "A4+_show_scada" := "A4+";
END_REGION

REGION Network 15: PLC-->PLC
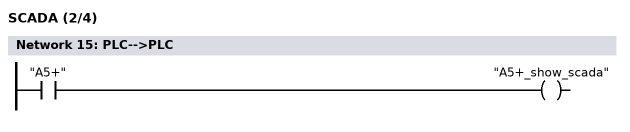
   RUNG wire#powerrail
      Contact( "A5+" )
      Coil( "A5+_show_scada" )
   END_RUNG
   // the same network as SCL:
   "A5+_show_scada" := "A5+";
END_REGION

REGION Network 16: PID PARAMETERS FROM THE SCADA
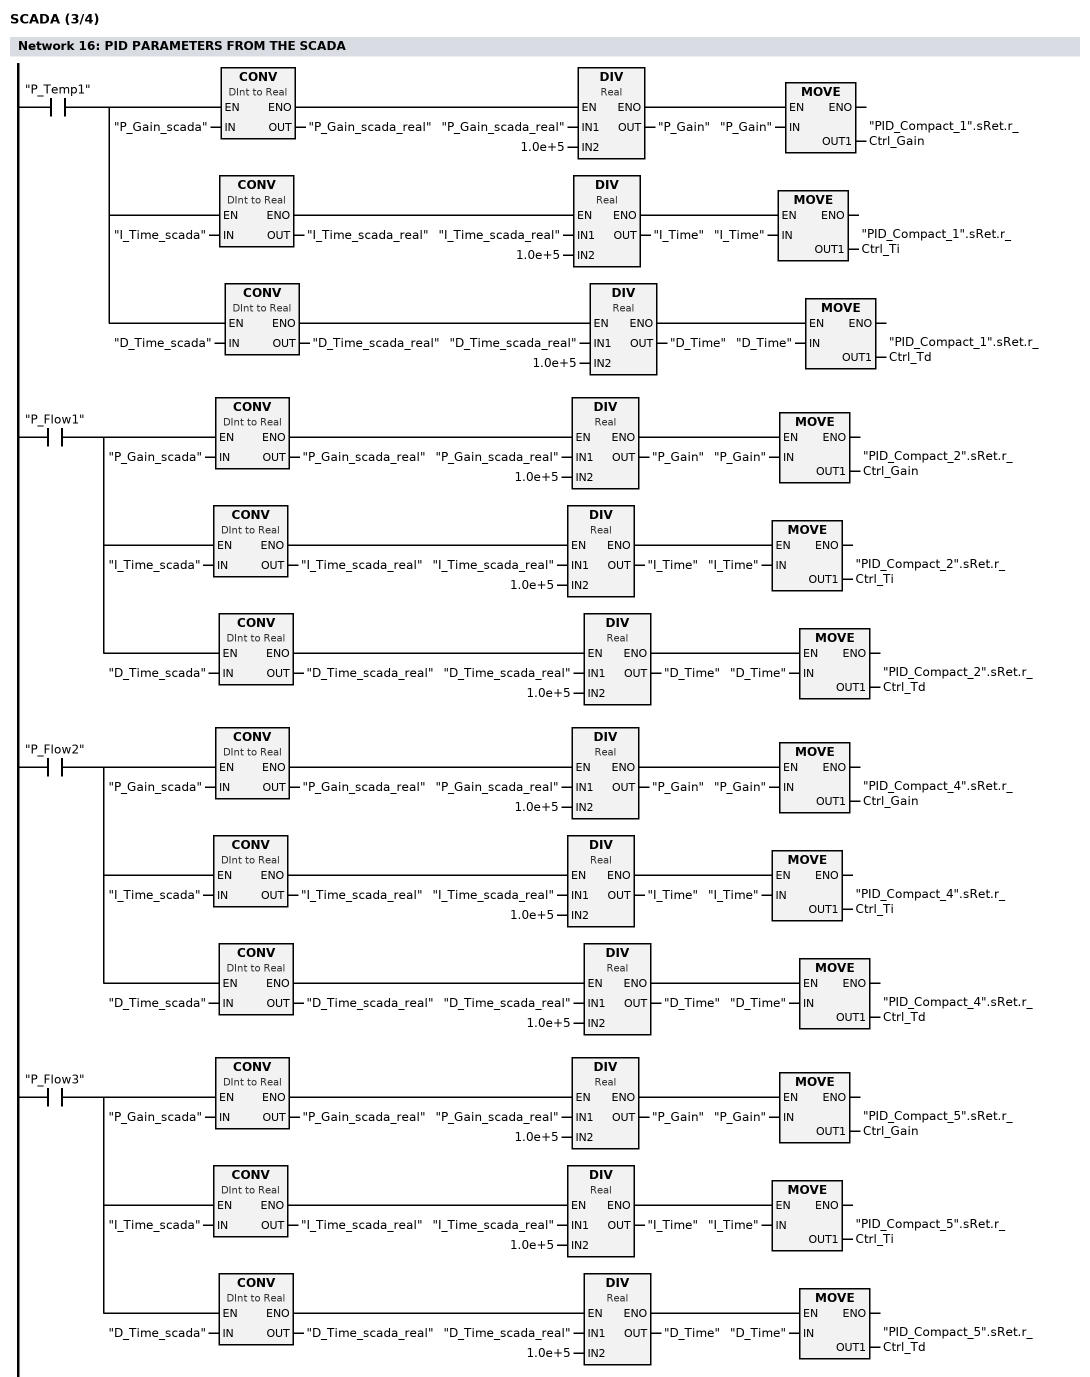
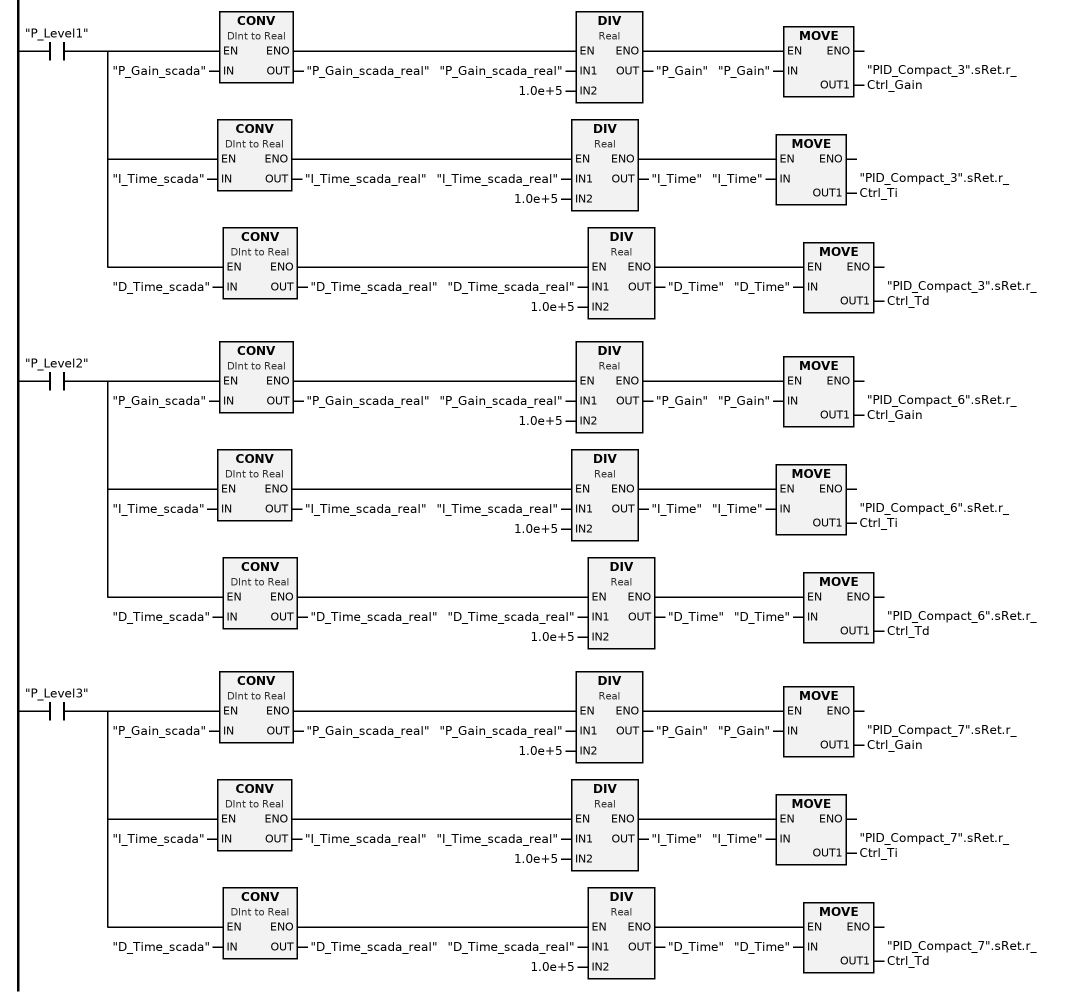
   RUNG wire#powerrail
      Contact( "P_Temp1" )
      wire#w1
      { S7_Templates := "[SrcType := DInt, DestType := Real]"; S7_GenerateENO := "TRUE" } Convert(in := "P_Gain_scada", out => "P_Gain_scada_real")
      { S7_Templates := "SrcType := Real"; S7_GenerateENO := "TRUE" } Div(in1 := "P_Gain_scada_real", in2 := 1.0e+5, out => "P_Gain")
      { S7_GenerateENO := "TRUE" } Move(in := "P_Gain", out1 => "PID_Compact_1".sRet.r_Ctrl_Gain)
   END_RUNG
   RUNG wire#w1
      { S7_Templates := "[SrcType := DInt, DestType := Real]"; S7_GenerateENO := "TRUE" } Convert(in := "I_Time_scada", out => "I_Time_scada_real")
      { S7_Templates := "SrcType := Real"; S7_GenerateENO := "TRUE" } Div(in1 := "I_Time_scada_real", in2 := 1.0e+5, out => "I_Time")
      { S7_GenerateENO := "TRUE" } Move(in := "I_Time", out1 => "PID_Compact_1".sRet.r_Ctrl_Ti)
   END_RUNG
   RUNG wire#w1
      { S7_Templates := "[SrcType := DInt, DestType := Real]"; S7_GenerateENO := "TRUE" } Convert(in := "D_Time_scada", out => "D_Time_scada_real")
      { S7_Templates := "SrcType := Real"; S7_GenerateENO := "TRUE" } Div(in1 := "D_Time_scada_real", in2 := 1.0e+5, out => "D_Time")
      { S7_GenerateENO := "TRUE" } Move(in := "D_Time", out1 => "PID_Compact_1".sRet.r_Ctrl_Td)
   END_RUNG
   RUNG wire#powerrail
      Contact( "P_Flow1" )
      wire#w2
      { S7_Templates := "[SrcType := DInt, DestType := Real]"; S7_GenerateENO := "TRUE" } Convert(in := "P_Gain_scada", out => "P_Gain_scada_real")
      { S7_Templates := "SrcType := Real"; S7_GenerateENO := "TRUE" } Div(in1 := "P_Gain_scada_real", in2 := 1.0e+5, out => "P_Gain")
      { S7_GenerateENO := "TRUE" } Move(in := "P_Gain", out1 => "PID_Compact_2".sRet.r_Ctrl_Gain)
   END_RUNG
   RUNG wire#w2
      { S7_Templates := "[SrcType := DInt, DestType := Real]"; S7_GenerateENO := "TRUE" } Convert(in := "I_Time_scada", out => "I_Time_scada_real")
      { S7_Templates := "SrcType := Real"; S7_GenerateENO := "TRUE" } Div(in1 := "I_Time_scada_real", in2 := 1.0e+5, out => "I_Time")
      { S7_GenerateENO := "TRUE" } Move(in := "I_Time", out1 => "PID_Compact_2".sRet.r_Ctrl_Ti)
   END_RUNG
   RUNG wire#w2
      { S7_Templates := "[SrcType := DInt, DestType := Real]"; S7_GenerateENO := "TRUE" } Convert(in := "D_Time_scada", out => "D_Time_scada_real")
      { S7_Templates := "SrcType := Real"; S7_GenerateENO := "TRUE" } Div(in1 := "D_Time_scada_real", in2 := 1.0e+5, out => "D_Time")
      { S7_GenerateENO := "TRUE" } Move(in := "D_Time", out1 => "PID_Compact_2".sRet.r_Ctrl_Td)
   END_RUNG
   RUNG wire#powerrail
      Contact( "P_Flow2" )
      wire#w3
      { S7_Templates := "[SrcType := DInt, DestType := Real]"; S7_GenerateENO := "TRUE" } Convert(in := "P_Gain_scada", out => "P_Gain_scada_real")
      { S7_Templates := "SrcType := Real"; S7_GenerateENO := "TRUE" } Div(in1 := "P_Gain_scada_real", in2 := 1.0e+5, out => "P_Gain")
      { S7_GenerateENO := "TRUE" } Move(in := "P_Gain", out1 => "PID_Compact_4".sRet.r_Ctrl_Gain)
   END_RUNG
   RUNG wire#w3
      { S7_Templates := "[SrcType := DInt, DestType := Real]"; S7_GenerateENO := "TRUE" } Convert(in := "I_Time_scada", out => "I_Time_scada_real")
      { S7_Templates := "SrcType := Real"; S7_GenerateENO := "TRUE" } Div(in1 := "I_Time_scada_real", in2 := 1.0e+5, out => "I_Time")
      { S7_GenerateENO := "TRUE" } Move(in := "I_Time", out1 => "PID_Compact_4".sRet.r_Ctrl_Ti)
   END_RUNG
   RUNG wire#w3
      { S7_Templates := "[SrcType := DInt, DestType := Real]"; S7_GenerateENO := "TRUE" } Convert(in := "D_Time_scada", out => "D_Time_scada_real")
      { S7_Templates := "SrcType := Real"; S7_GenerateENO := "TRUE" } Div(in1 := "D_Time_scada_real", in2 := 1.0e+5, out => "D_Time")
      { S7_GenerateENO := "TRUE" } Move(in := "D_Time", out1 => "PID_Compact_4".sRet.r_Ctrl_Td)
   END_RUNG
   RUNG wire#powerrail
      Contact( "P_Flow3" )
      wire#w4
      { S7_Templates := "[SrcType := DInt, DestType := Real]"; S7_GenerateENO := "TRUE" } Convert(in := "P_Gain_scada", out => "P_Gain_scada_real")
      { S7_Templates := "SrcType := Real"; S7_GenerateENO := "TRUE" } Div(in1 := "P_Gain_scada_real", in2 := 1.0e+5, out => "P_Gain")
      { S7_GenerateENO := "TRUE" } Move(in := "P_Gain", out1 => "PID_Compact_5".sRet.r_Ctrl_Gain)
   END_RUNG
   RUNG wire#w4
      { S7_Templates := "[SrcType := DInt, DestType := Real]"; S7_GenerateENO := "TRUE" } Convert(in := "I_Time_scada", out => "I_Time_scada_real")
      { S7_Templates := "SrcType := Real"; S7_GenerateENO := "TRUE" } Div(in1 := "I_Time_scada_real", in2 := 1.0e+5, out => "I_Time")
      { S7_GenerateENO := "TRUE" } Move(in := "I_Time", out1 => "PID_Compact_5".sRet.r_Ctrl_Ti)
   END_RUNG
   RUNG wire#w4
      { S7_Templates := "[SrcType := DInt, DestType := Real]"; S7_GenerateENO := "TRUE" } Convert(in := "D_Time_scada", out => "D_Time_scada_real")
      { S7_Templates := "SrcType := Real"; S7_GenerateENO := "TRUE" } Div(in1 := "D_Time_scada_real", in2 := 1.0e+5, out => "D_Time")
      { S7_GenerateENO := "TRUE" } Move(in := "D_Time", out1 => "PID_Compact_5".sRet.r_Ctrl_Td)
   END_RUNG
   RUNG wire#powerrail
      Contact( "P_Level1" )
      wire#w5
      { S7_Templates := "[SrcType := DInt, DestType := Real]"; S7_GenerateENO := "TRUE" } Convert(in := "P_Gain_scada", out => "P_Gain_scada_real")
      { S7_Templates := "SrcType := Real"; S7_GenerateENO := "TRUE" } Div(in1 := "P_Gain_scada_real", in2 := 1.0e+5, out => "P_Gain")
      { S7_GenerateENO := "TRUE" } Move(in := "P_Gain", out1 => "PID_Compact_3".sRet.r_Ctrl_Gain)
   END_RUNG
   RUNG wire#w5
      { S7_Templates := "[SrcType := DInt, DestType := Real]"; S7_GenerateENO := "TRUE" } Convert(in := "I_Time_scada", out => "I_Time_scada_real")
      { S7_Templates := "SrcType := Real"; S7_GenerateENO := "TRUE" } Div(in1 := "I_Time_scada_real", in2 := 1.0e+5, out => "I_Time")
      { S7_GenerateENO := "TRUE" } Move(in := "I_Time", out1 => "PID_Compact_3".sRet.r_Ctrl_Ti)
   END_RUNG
   RUNG wire#w5
      { S7_Templates := "[SrcType := DInt, DestType := Real]"; S7_GenerateENO := "TRUE" } Convert(in := "D_Time_scada", out => "D_Time_scada_real")
      { S7_Templates := "SrcType := Real"; S7_GenerateENO := "TRUE" } Div(in1 := "D_Time_scada_real", in2 := 1.0e+5, out => "D_Time")
      { S7_GenerateENO := "TRUE" } Move(in := "D_Time", out1 => "PID_Compact_3".sRet.r_Ctrl_Td)
   END_RUNG
   RUNG wire#powerrail
      Contact( "P_Level2" )
      wire#w6
      { S7_Templates := "[SrcType := DInt, DestType := Real]"; S7_GenerateENO := "TRUE" } Convert(in := "P_Gain_scada", out => "P_Gain_scada_real")
      { S7_Templates := "SrcType := Real"; S7_GenerateENO := "TRUE" } Div(in1 := "P_Gain_scada_real", in2 := 1.0e+5, out => "P_Gain")
      { S7_GenerateENO := "TRUE" } Move(in := "P_Gain", out1 => "PID_Compact_6".sRet.r_Ctrl_Gain)
   END_RUNG
   RUNG wire#w6
      { S7_Templates := "[SrcType := DInt, DestType := Real]"; S7_GenerateENO := "TRUE" } Convert(in := "I_Time_scada", out => "I_Time_scada_real")
      { S7_Templates := "SrcType := Real"; S7_GenerateENO := "TRUE" } Div(in1 := "I_Time_scada_real", in2 := 1.0e+5, out => "I_Time")
      { S7_GenerateENO := "TRUE" } Move(in := "I_Time", out1 => "PID_Compact_6".sRet.r_Ctrl_Ti)
   END_RUNG
   RUNG wire#w6
      { S7_Templates := "[SrcType := DInt, DestType := Real]"; S7_GenerateENO := "TRUE" } Convert(in := "D_Time_scada", out => "D_Time_scada_real")
      { S7_Templates := "SrcType := Real"; S7_GenerateENO := "TRUE" } Div(in1 := "D_Time_scada_real", in2 := 1.0e+5, out => "D_Time")
      { S7_GenerateENO := "TRUE" } Move(in := "D_Time", out1 => "PID_Compact_6".sRet.r_Ctrl_Td)
   END_RUNG
   RUNG wire#powerrail
      Contact( "P_Level3" )
      wire#w7
      { S7_Templates := "[SrcType := DInt, DestType := Real]"; S7_GenerateENO := "TRUE" } Convert(in := "P_Gain_scada", out => "P_Gain_scada_real")
      { S7_Templates := "SrcType := Real"; S7_GenerateENO := "TRUE" } Div(in1 := "P_Gain_scada_real", in2 := 1.0e+5, out => "P_Gain")
      { S7_GenerateENO := "TRUE" } Move(in := "P_Gain", out1 => "PID_Compact_7".sRet.r_Ctrl_Gain)
   END_RUNG
   RUNG wire#w7
      { S7_Templates := "[SrcType := DInt, DestType := Real]"; S7_GenerateENO := "TRUE" } Convert(in := "I_Time_scada", out => "I_Time_scada_real")
      { S7_Templates := "SrcType := Real"; S7_GenerateENO := "TRUE" } Div(in1 := "I_Time_scada_real", in2 := 1.0e+5, out => "I_Time")
      { S7_GenerateENO := "TRUE" } Move(in := "I_Time", out1 => "PID_Compact_7".sRet.r_Ctrl_Ti)
   END_RUNG
   RUNG wire#w7
      { S7_Templates := "[SrcType := DInt, DestType := Real]"; S7_GenerateENO := "TRUE" } Convert(in := "D_Time_scada", out => "D_Time_scada_real")
      { S7_Templates := "SrcType := Real"; S7_GenerateENO := "TRUE" } Div(in1 := "D_Time_scada_real", in2 := 1.0e+5, out => "D_Time")
      { S7_GenerateENO := "TRUE" } Move(in := "D_Time", out1 => "PID_Compact_7".sRet.r_Ctrl_Td)
   END_RUNG
   // the same network as SCL:
   // ENO of a box is taken as its EN; it also drops when the box reports an error
   IF "P_Temp1" THEN
       "P_Gain_scada_real" := DINT_TO_REAL("P_Gain_scada");
       "P_Gain" := "P_Gain_scada_real" / 1.0e+5;
       "PID_Compact_1".sRet.r_Ctrl_Gain := "P_Gain";
       "I_Time_scada_real" := DINT_TO_REAL("I_Time_scada");
       "I_Time" := "I_Time_scada_real" / 1.0e+5;
       "PID_Compact_1".sRet.r_Ctrl_Ti := "I_Time";
       "D_Time_scada_real" := DINT_TO_REAL("D_Time_scada");
       "D_Time" := "D_Time_scada_real" / 1.0e+5;
       "PID_Compact_1".sRet.r_Ctrl_Td := "D_Time";
   END_IF;
   IF "P_Flow1" THEN
       "P_Gain_scada_real" := DINT_TO_REAL("P_Gain_scada");
       "P_Gain" := "P_Gain_scada_real" / 1.0e+5;
       "PID_Compact_2".sRet.r_Ctrl_Gain := "P_Gain";
       "I_Time_scada_real" := DINT_TO_REAL("I_Time_scada");
       "I_Time" := "I_Time_scada_real" / 1.0e+5;
       "PID_Compact_2".sRet.r_Ctrl_Ti := "I_Time";
       "D_Time_scada_real" := DINT_TO_REAL("D_Time_scada");
       "D_Time" := "D_Time_scada_real" / 1.0e+5;
       "PID_Compact_2".sRet.r_Ctrl_Td := "D_Time";
   END_IF;
   IF "P_Flow2" THEN
       "P_Gain_scada_real" := DINT_TO_REAL("P_Gain_scada");
       "P_Gain" := "P_Gain_scada_real" / 1.0e+5;
       "PID_Compact_4".sRet.r_Ctrl_Gain := "P_Gain";
       "I_Time_scada_real" := DINT_TO_REAL("I_Time_scada");
       "I_Time" := "I_Time_scada_real" / 1.0e+5;
       "PID_Compact_4".sRet.r_Ctrl_Ti := "I_Time";
       "D_Time_scada_real" := DINT_TO_REAL("D_Time_scada");
       "D_Time" := "D_Time_scada_real" / 1.0e+5;
       "PID_Compact_4".sRet.r_Ctrl_Td := "D_Time";
   END_IF;
   IF "P_Flow3" THEN
       "P_Gain_scada_real" := DINT_TO_REAL("P_Gain_scada");
       "P_Gain" := "P_Gain_scada_real" / 1.0e+5;
       "PID_Compact_5".sRet.r_Ctrl_Gain := "P_Gain";
       "I_Time_scada_real" := DINT_TO_REAL("I_Time_scada");
       "I_Time" := "I_Time_scada_real" / 1.0e+5;
       "PID_Compact_5".sRet.r_Ctrl_Ti := "I_Time";
       "D_Time_scada_real" := DINT_TO_REAL("D_Time_scada");
       "D_Time" := "D_Time_scada_real" / 1.0e+5;
       "PID_Compact_5".sRet.r_Ctrl_Td := "D_Time";
   END_IF;
   IF "P_Level1" THEN
       "P_Gain_scada_real" := DINT_TO_REAL("P_Gain_scada");
       "P_Gain" := "P_Gain_scada_real" / 1.0e+5;
       "PID_Compact_3".sRet.r_Ctrl_Gain := "P_Gain";
       "I_Time_scada_real" := DINT_TO_REAL("I_Time_scada");
       "I_Time" := "I_Time_scada_real" / 1.0e+5;
       "PID_Compact_3".sRet.r_Ctrl_Ti := "I_Time";
       "D_Time_scada_real" := DINT_TO_REAL("D_Time_scada");
       "D_Time" := "D_Time_scada_real" / 1.0e+5;
       "PID_Compact_3".sRet.r_Ctrl_Td := "D_Time";
   END_IF;
   IF "P_Level2" THEN
       "P_Gain_scada_real" := DINT_TO_REAL("P_Gain_scada");
       "P_Gain" := "P_Gain_scada_real" / 1.0e+5;
       "PID_Compact_6".sRet.r_Ctrl_Gain := "P_Gain";
       "I_Time_scada_real" := DINT_TO_REAL("I_Time_scada");
       "I_Time" := "I_Time_scada_real" / 1.0e+5;
       "PID_Compact_6".sRet.r_Ctrl_Ti := "I_Time";
       "D_Time_scada_real" := DINT_TO_REAL("D_Time_scada");
       "D_Time" := "D_Time_scada_real" / 1.0e+5;
       "PID_Compact_6".sRet.r_Ctrl_Td := "D_Time";
   END_IF;
   IF "P_Level3" THEN
       "P_Gain_scada_real" := DINT_TO_REAL("P_Gain_scada");
       "P_Gain" := "P_Gain_scada_real" / 1.0e+5;
       "PID_Compact_7".sRet.r_Ctrl_Gain := "P_Gain";
       "I_Time_scada_real" := DINT_TO_REAL("I_Time_scada");
       "I_Time" := "I_Time_scada_real" / 1.0e+5;
       "PID_Compact_7".sRet.r_Ctrl_Ti := "I_Time";
       "D_Time_scada_real" := DINT_TO_REAL("D_Time_scada");
       "D_Time" := "D_Time_scada_real" / 1.0e+5;
       "PID_Compact_7".sRet.r_Ctrl_Td := "D_Time";
   END_IF;
END_REGION

REGION Network 17: SEND CONTROL VALUE TO THE SCADA
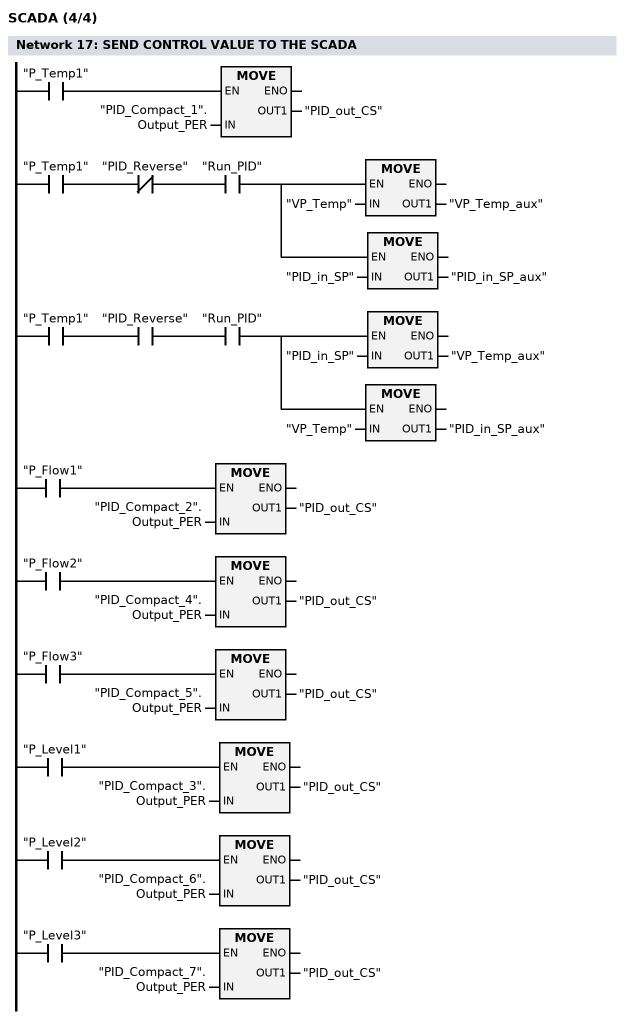
   RUNG wire#powerrail
      Contact( "P_Temp1" )
      { S7_GenerateENO := "TRUE" } Move(in := "PID_Compact_1".Output_PER, out1 => "PID_out_CS")
   END_RUNG
   RUNG wire#powerrail
      Contact( "P_Temp1" )
      I_Contact( "PID_Reverse" )
      Contact( "Run_PID" )
      wire#w1
      { S7_GenerateENO := "TRUE" } Move(in := "VP_Temp", out1 => "VP_Temp_aux")
   END_RUNG
   RUNG wire#w1
      { S7_GenerateENO := "TRUE" } Move(in := "PID_in_SP", out1 => "PID_in_SP_aux")
   END_RUNG
   RUNG wire#powerrail
      Contact( "P_Temp1" )
      Contact( "PID_Reverse" )
      Contact( "Run_PID" )
      wire#w2
      { S7_GenerateENO := "TRUE" } Move(in := "PID_in_SP", out1 => "VP_Temp_aux")
   END_RUNG
   RUNG wire#w2
      { S7_GenerateENO := "TRUE" } Move(in := "VP_Temp", out1 => "PID_in_SP_aux")
   END_RUNG
   RUNG wire#powerrail
      Contact( "P_Flow1" )
      { S7_GenerateENO := "TRUE" } Move(in := "PID_Compact_2".Output_PER, out1 => "PID_out_CS")
   END_RUNG
   RUNG wire#powerrail
      Contact( "P_Flow2" )
      { S7_GenerateENO := "TRUE" } Move(in := "PID_Compact_4".Output_PER, out1 => "PID_out_CS")
   END_RUNG
   RUNG wire#powerrail
      Contact( "P_Flow3" )
      { S7_GenerateENO := "TRUE" } Move(in := "PID_Compact_5".Output_PER, out1 => "PID_out_CS")
   END_RUNG
   RUNG wire#powerrail
      Contact( "P_Level1" )
      { S7_GenerateENO := "TRUE" } Move(in := "PID_Compact_3".Output_PER, out1 => "PID_out_CS")
   END_RUNG
   RUNG wire#powerrail
      Contact( "P_Level2" )
      { S7_GenerateENO := "TRUE" } Move(in := "PID_Compact_6".Output_PER, out1 => "PID_out_CS")
   END_RUNG
   RUNG wire#powerrail
      Contact( "P_Level3" )
      { S7_GenerateENO := "TRUE" } Move(in := "PID_Compact_7".Output_PER, out1 => "PID_out_CS")
   END_RUNG
   // the same network as SCL:
   IF "P_Temp1" THEN "PID_out_CS" := "PID_Compact_1".Output_PER; END_IF;
   IF "P_Temp1" AND NOT "PID_Reverse" AND "Run_PID" THEN
       "VP_Temp_aux" := "VP_Temp";
       "PID_in_SP_aux" := "PID_in_SP";
   END_IF;
   IF "P_Temp1" AND "PID_Reverse" AND "Run_PID" THEN
       "VP_Temp_aux" := "PID_in_SP";
       "PID_in_SP_aux" := "VP_Temp";
   END_IF;
   IF "P_Flow1" THEN "PID_out_CS" := "PID_Compact_2".Output_PER; END_IF;
   IF "P_Flow2" THEN "PID_out_CS" := "PID_Compact_4".Output_PER; END_IF;
   IF "P_Flow3" THEN "PID_out_CS" := "PID_Compact_5".Output_PER; END_IF;
   IF "P_Level1" THEN "PID_out_CS" := "PID_Compact_3".Output_PER; END_IF;
   IF "P_Level2" THEN "PID_out_CS" := "PID_Compact_6".Output_PER; END_IF;
   IF "P_Level3" THEN "PID_out_CS" := "PID_Compact_7".Output_PER; END_IF;
END_REGION
END_FUNCTION

FUNCTION "OUTPUTS" : Void   // FC4, LAD
TITLE = OUTPUTS FROM THE PLC
{ S7_Optimized_Access := 'TRUE' }
VERSION : 0.1
BEGIN

REGION Network 1: A4+
   // Opening of the output solenoid of the AUXILIARY TANK
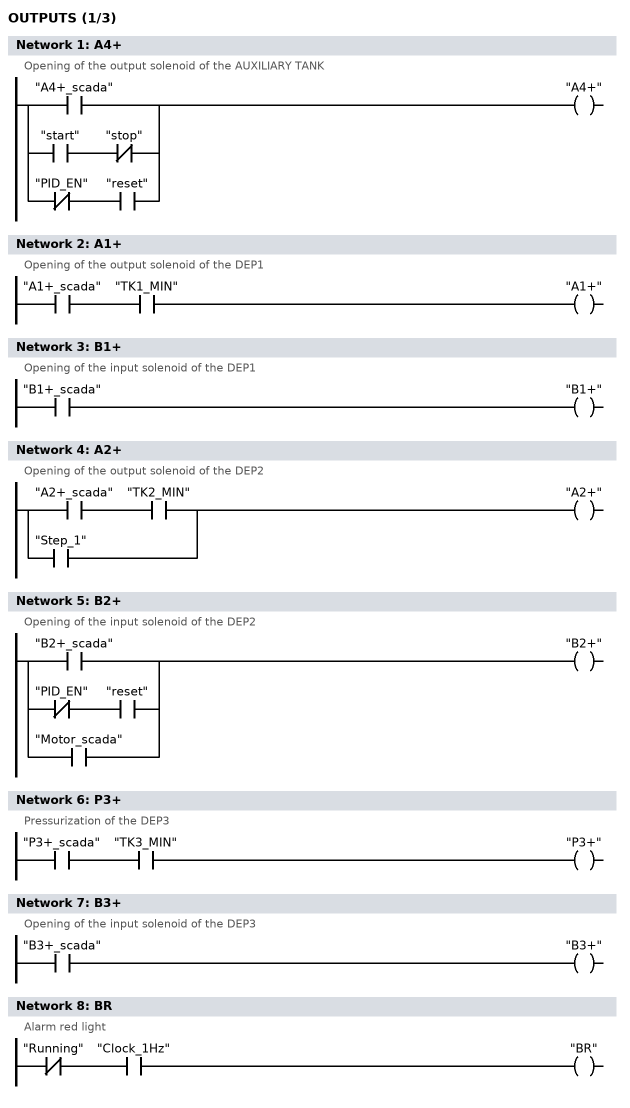
   RUNG wire#powerrail
      Contact( "A4+_scada" )
      wire#w1
      Coil( "A4+" )
   END_RUNG
   RUNG wire#powerrail
      Contact( "start" )
      I_Contact( "stop" )
   END_RUNG wire#w1
   RUNG wire#powerrail
      I_Contact( "PID_EN" )
      Contact( "reset" )
   END_RUNG wire#w1
   // the same network as SCL:
   "A4+" := "A4+_scada" OR ("start" AND NOT "stop") OR (NOT "PID_EN" AND "reset");
END_REGION

REGION Network 2: A1+
   // Opening of the output solenoid of the DEP1
   RUNG wire#powerrail
      Contact( "A1+_scada" )
      Contact( "TK1_MIN" )
      Coil( "A1+" )
   END_RUNG
   // the same network as SCL:
   "A1+" := "A1+_scada" AND "TK1_MIN";
END_REGION

REGION Network 3: B1+
   // Opening of the input solenoid of the DEP1
   RUNG wire#powerrail
      Contact( "B1+_scada" )
      Coil( "B1+" )
   END_RUNG
   // the same network as SCL:
   "B1+" := "B1+_scada";
END_REGION

REGION Network 4: A2+
   // Opening of the output solenoid of the DEP2
   RUNG wire#powerrail
      Contact( "A2+_scada" )
      Contact( "TK2_MIN" )
      wire#w1
      Coil( "A2+" )
   END_RUNG
   RUNG wire#powerrail
      Contact( "Step_1" )
   END_RUNG wire#w1
   // the same network as SCL:
   "A2+" := ("A2+_scada" AND "TK2_MIN") OR "Step_1";
END_REGION

REGION Network 5: B2+
   // Opening of the input solenoid of the DEP2
   RUNG wire#powerrail
      Contact( "B2+_scada" )
      wire#w1
      Coil( "B2+" )
   END_RUNG
   RUNG wire#powerrail
      I_Contact( "PID_EN" )
      Contact( "reset" )
   END_RUNG wire#w1
   RUNG wire#powerrail
      Contact( "Motor_scada" )
   END_RUNG wire#w1
   // the same network as SCL:
   "B2+" := "B2+_scada" OR (NOT "PID_EN" AND "reset") OR "Motor_scada";
END_REGION

REGION Network 6: P3+
   // Pressurization of the DEP3
   RUNG wire#powerrail
      Contact( "P3+_scada" )
      Contact( "TK3_MIN" )
      Coil( "P3+" )
   END_RUNG
   // the same network as SCL:
   "P3+" := "P3+_scada" AND "TK3_MIN";
END_REGION

REGION Network 7: B3+
   // Opening of the input solenoid of the DEP3
   RUNG wire#powerrail
      Contact( "B3+_scada" )
      Coil( "B3+" )
   END_RUNG
   // the same network as SCL:
   "B3+" := "B3+_scada";
END_REGION

REGION Network 8: BR
   // Alarm red light
   RUNG wire#powerrail
      I_Contact( "Running" )
      Contact( "Clock_1Hz" )
      Coil( "BR" )
   END_RUNG
   // the same network as SCL:
   "BR" := NOT "Running" AND "Clock_1Hz";
END_REGION

REGION Network 9: Invert_VBus
   // Polarity change of the Peltier cells and activation of the fan
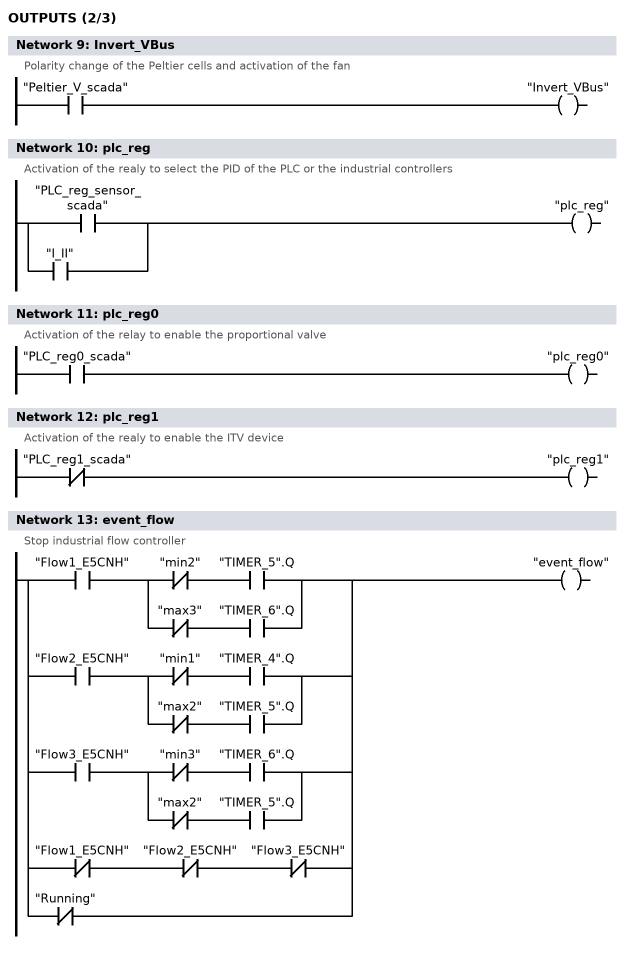
   RUNG wire#powerrail
      Contact( "Peltier_V_scada" )
      Coil( "Invert_VBus" )
   END_RUNG
   // the same network as SCL:
   "Invert_VBus" := "Peltier_V_scada";
END_REGION

REGION Network 10: plc_reg
   // Activation of the realy to select the PID of the PLC or the industrial controllers
   RUNG wire#powerrail
      Contact( "PLC_reg_sensor_scada" )
      wire#w1
      Coil( "plc_reg" )
   END_RUNG
   RUNG wire#powerrail
      Contact( "I_II" )
   END_RUNG wire#w1
   // the same network as SCL:
   "plc_reg" := "PLC_reg_sensor_scada" OR "I_II";
END_REGION

REGION Network 11: plc_reg0
   // Activation of the relay to enable the proportional valve
   RUNG wire#powerrail
      Contact( "PLC_reg0_scada" )
      Coil( "plc_reg0" )
   END_RUNG
   // the same network as SCL:
   "plc_reg0" := "PLC_reg0_scada";
END_REGION

REGION Network 12: plc_reg1
   // Activation of the realy to enable the ITV device
   RUNG wire#powerrail
      I_Contact( "PLC_reg1_scada" )
      Coil( "plc_reg1" )
   END_RUNG
   // the same network as SCL:
   "plc_reg1" := NOT "PLC_reg1_scada";
END_REGION

REGION Network 13: event_flow
   // Stop industrial flow controller
   RUNG wire#powerrail
      Contact( "Flow1_E5CNH" )
      wire#w1
      I_Contact( "min2" )
      Contact( "TIMER_5".Q )
      wire#w2
      Coil( "event_flow" )
   END_RUNG
   RUNG wire#w1
      I_Contact( "max3" )
      Contact( "TIMER_6".Q )
   END_RUNG wire#w2
   RUNG wire#powerrail
      Contact( "Flow2_E5CNH" )
      wire#w3
      I_Contact( "min1" )
      Contact( "TIMER_4".Q )
   END_RUNG wire#w2
   RUNG wire#w3
      I_Contact( "max2" )
      Contact( "TIMER_5".Q )
   END_RUNG wire#w2
   RUNG wire#powerrail
      Contact( "Flow3_E5CNH" )
      wire#w4
      I_Contact( "min3" )
      Contact( "TIMER_6".Q )
   END_RUNG wire#w2
   RUNG wire#w4
      I_Contact( "max2" )
      Contact( "TIMER_5".Q )
   END_RUNG wire#w2
   RUNG wire#powerrail
      I_Contact( "Flow1_E5CNH" )
      I_Contact( "Flow2_E5CNH" )
      I_Contact( "Flow3_E5CNH" )
   END_RUNG wire#w2
   RUNG wire#powerrail
      I_Contact( "Running" )
   END_RUNG wire#w2
   // the same network as SCL:
   "event_flow" := ("Flow1_E5CNH" AND ((NOT "min2" AND "TIMER_5".Q) OR (NOT "max3" AND "TIMER_6".Q))) OR ("Flow2_E5CNH" AND ((NOT "min1" AND "TIMER_4".Q) OR (NOT "max2" AND "TIMER_5".Q))) OR ("Flow3_E5CNH" AND ((NOT "min3" AND "TIMER_6".Q) OR (NOT "max2" AND "TIMER_5".Q))) OR (NOT "Flow1_E5CNH" AND NOT "Flow2_E5CNH" AND NOT "Flow3_E5CNH") OR NOT "Running";
END_REGION

REGION Network 14: event_level
   // Stop industrial level controller
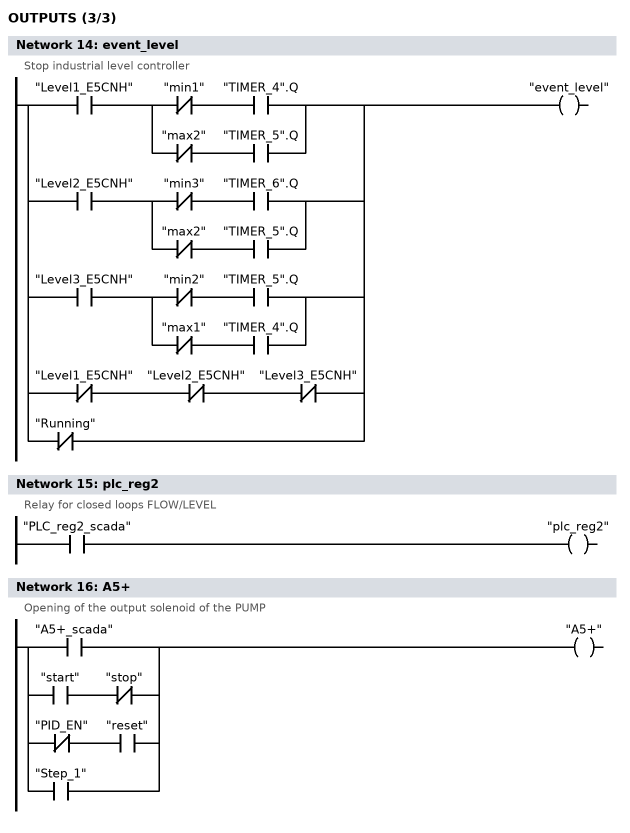
   RUNG wire#powerrail
      Contact( "Level1_E5CNH" )
      wire#w1
      I_Contact( "min1" )
      Contact( "TIMER_4".Q )
      wire#w2
      Coil( "event_level" )
   END_RUNG
   RUNG wire#w1
      I_Contact( "max2" )
      Contact( "TIMER_5".Q )
   END_RUNG wire#w2
   RUNG wire#powerrail
      Contact( "Level2_E5CNH" )
      wire#w3
      I_Contact( "min3" )
      Contact( "TIMER_6".Q )
   END_RUNG wire#w2
   RUNG wire#w3
      I_Contact( "max2" )
      Contact( "TIMER_5".Q )
   END_RUNG wire#w2
   RUNG wire#powerrail
      Contact( "Level3_E5CNH" )
      wire#w4
      I_Contact( "min2" )
      Contact( "TIMER_5".Q )
   END_RUNG wire#w2
   RUNG wire#w4
      I_Contact( "max1" )
      Contact( "TIMER_4".Q )
   END_RUNG wire#w2
   RUNG wire#powerrail
      I_Contact( "Level1_E5CNH" )
      I_Contact( "Level2_E5CNH" )
      I_Contact( "Level3_E5CNH" )
   END_RUNG wire#w2
   RUNG wire#powerrail
      I_Contact( "Running" )
   END_RUNG wire#w2
   // the same network as SCL:
   "event_level" := ("Level1_E5CNH" AND ((NOT "min1" AND "TIMER_4".Q) OR (NOT "max2" AND "TIMER_5".Q))) OR ("Level2_E5CNH" AND ((NOT "min3" AND "TIMER_6".Q) OR (NOT "max2" AND "TIMER_5".Q))) OR ("Level3_E5CNH" AND ((NOT "min2" AND "TIMER_5".Q) OR (NOT "max1" AND "TIMER_4".Q))) OR (NOT "Level1_E5CNH" AND NOT "Level2_E5CNH" AND NOT "Level3_E5CNH") OR NOT "Running";
END_REGION

REGION Network 15: plc_reg2
   // Relay for closed loops FLOW/LEVEL
   RUNG wire#powerrail
      Contact( "PLC_reg2_scada" )
      Coil( "plc_reg2" )
   END_RUNG
   // the same network as SCL:
   "plc_reg2" := "PLC_reg2_scada";
END_REGION

REGION Network 16: A5+
   // Opening of the output solenoid of the PUMP
   RUNG wire#powerrail
      Contact( "A5+_scada" )
      wire#w1
      Coil( "A5+" )
   END_RUNG
   RUNG wire#powerrail
      Contact( "start" )
      I_Contact( "stop" )
   END_RUNG wire#w1
   RUNG wire#powerrail
      I_Contact( "PID_EN" )
      Contact( "reset" )
   END_RUNG wire#w1
   RUNG wire#powerrail
      Contact( "Step_1" )
   END_RUNG wire#w1
   // the same network as SCL:
   "A5+" := "A5+_scada" OR ("start" AND NOT "stop") OR (NOT "PID_EN" AND "reset") OR "Step_1";
END_REGION
END_FUNCTION

FUNCTION "COMMUNICATIONS" : Void   // FC5, LAD
TITLE = COMMUNICATION WITH IPC202 AND IPC203
{ S7_Optimized_Access := 'FALSE' }
VERSION : 0.1
BEGIN

REGION Network 1: GET function (reading from the IPC202)
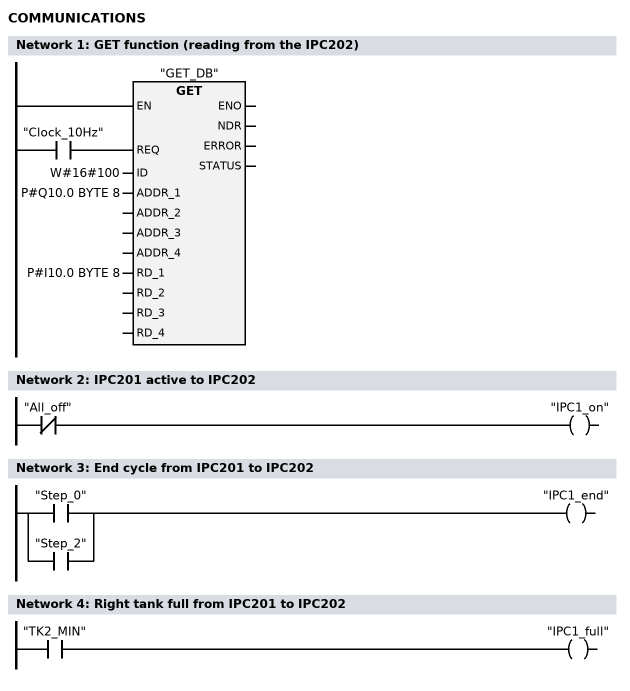
   "GET_DB"(REQ := "Clock_10Hz", ID := W#16#100, ADDR_1 := P#Q10.0 BYTE 8, RD_1 := P#I10.0 BYTE 8);   // GET
END_REGION

REGION Network 2: IPC201 active to IPC202
   RUNG wire#powerrail
      I_Contact( "All_off" )
      Coil( "IPC1_on" )
   END_RUNG
   // the same network as SCL:
   "IPC1_on" := NOT "All_off";
END_REGION

REGION Network 3: End cycle from IPC201 to IPC202
   RUNG wire#powerrail
      Contact( "Step_0" )
      wire#w1
      Coil( "IPC1_end" )
   END_RUNG
   RUNG wire#powerrail
      Contact( "Step_2" )
   END_RUNG wire#w1
   // the same network as SCL:
   "IPC1_end" := "Step_0" OR "Step_2";
END_REGION

REGION Network 4: Right tank full from IPC201 to IPC202
   RUNG wire#powerrail
      Contact( "TK2_MIN" )
      Coil( "IPC1_full" )
   END_RUNG
   // the same network as SCL:
   "IPC1_full" := "TK2_MIN";
END_REGION
END_FUNCTION

FUNCTION "STEPS" : Void   // FC6, LAD
TITLE = STEPS
{ S7_Optimized_Access := 'TRUE' }
VERSION : 0.1
BEGIN

REGION Network 1: Step 0 - First step of the Grafcet
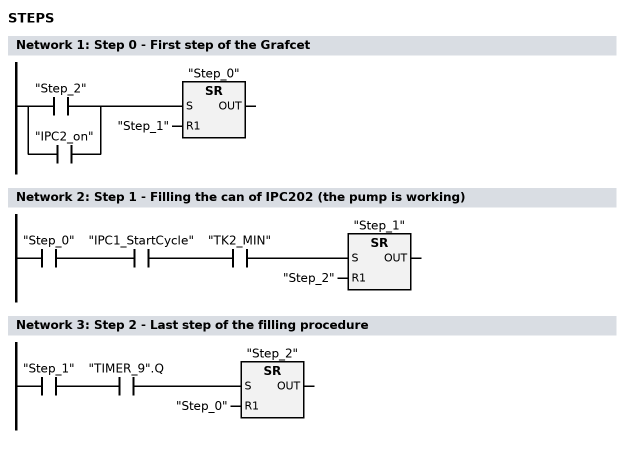
   RUNG wire#powerrail
      Contact( "Step_2" )
      wire#w1
      S_SR(operand := "Step_0", r1 := "Step_1")
   END_RUNG
   RUNG wire#powerrail
      Contact( "IPC2_on" )
   END_RUNG wire#w1
   // the same network as SCL:
   IF "Step_2" OR "IPC2_on" THEN
       "Step_0" := TRUE;   // SR flip-flop
   END_IF;
   IF "Step_1" THEN "Step_0" := FALSE; END_IF;
END_REGION

REGION Network 2: Step 1 - Filling the can of IPC202 (the pump is working)
   RUNG wire#powerrail
      Contact( "Step_0" )
      Contact( "IPC1_StartCycle" )
      Contact( "TK2_MIN" )
      S_SR(operand := "Step_1", r1 := "Step_2")
   END_RUNG
   // the same network as SCL:
   IF "Step_0" AND "IPC1_StartCycle" AND "TK2_MIN" THEN
       "Step_1" := TRUE;   // SR flip-flop
   END_IF;
   IF "Step_2" THEN "Step_1" := FALSE; END_IF;
END_REGION

REGION Network 3: Step 2 - Last step of the filling procedure
   RUNG wire#powerrail
      Contact( "Step_1" )
      Contact( "TIMER_9".Q )
      S_SR(operand := "Step_2", r1 := "Step_0")
   END_RUNG
   // the same network as SCL:
   IF "Step_1" AND "TIMER_9".Q THEN
       "Step_2" := TRUE;   // SR flip-flop
   END_IF;
   IF "Step_0" THEN "Step_2" := FALSE; END_IF;
END_REGION
END_FUNCTION

FUNCTION "PROGRAM" : Void   // FC7, LAD
{ S7_Optimized_Access := 'TRUE' }
VERSION : 0.1
   VAR_TEMP   // added for the SCL form of the ladder/FBD networks
      _w1 : Bool;
      _w2 : Bool;
      _w3 : Bool;
      _w4 : Bool;
      _w5 : Bool;
      _w6 : Bool;
   END_VAR
BEGIN

REGION Network 1: Program running and switch on for program
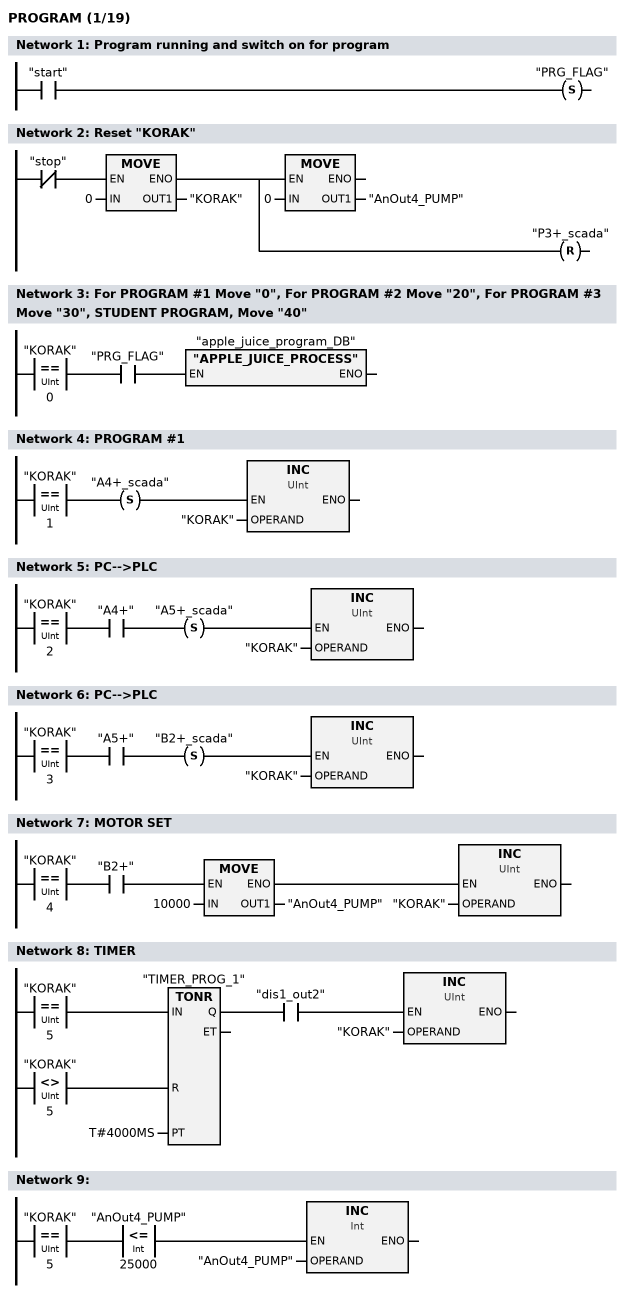
   RUNG wire#powerrail
      Contact( "start" )
      S_Coil( "PRG_FLAG" )
   END_RUNG
   // the same network as SCL:
   IF "start" THEN "PRG_FLAG" := TRUE; END_IF;
END_REGION

REGION Network 2: Reset "KORAK"
   RUNG wire#powerrail
      I_Contact( "stop" )
      Move(in := 0, out1 => "KORAK")
      wire#w1
      Move(in := 0, out1 => "AnOut4_PUMP")
   END_RUNG
   RUNG wire#w1
      R_Coil( "P3+_scada" )
   END_RUNG
   // the same network as SCL:
   IF NOT "stop" THEN
       "KORAK" := 0;
       "AnOut4_PUMP" := 0;
       "P3+_scada" := FALSE;
   END_IF;
END_REGION

REGION Network 3: For PROGRAM #1 Move "0", For PROGRAM #2 Move "20", For PROGRAM #3 Move "30", STUDENT PROGRAM, Move "40"
   RUNG wire#powerrail
      { S7_Templates := "SrcType := UInt" } EQ_Contact(in1 := "KORAK", in2 := 0)
      Contact( "PRG_FLAG" )
      "apple_juice_program_DB"()
   END_RUNG
   // the same network as SCL:
   IF ("KORAK" = 0) AND "PRG_FLAG" THEN
       "apple_juice_program_DB"();   // "APPLE_JUICE_PROCESS"
   END_IF;
END_REGION

REGION Network 4: PROGRAM #1
   RUNG wire#powerrail
      { S7_Templates := "SrcType := UInt" } EQ_Contact(in1 := "KORAK", in2 := 1)
      S_Coil( "A4+_scada" )
      { S7_Templates := "DestType := UInt" } Inc( "KORAK" )
   END_RUNG
   // the same network as SCL:
   IF "KORAK" = 1 THEN
       "A4+_scada" := TRUE;
       "KORAK" := "KORAK" + 1;
   END_IF;
END_REGION

REGION Network 5: PC-->PLC
   RUNG wire#powerrail
      { S7_Templates := "SrcType := UInt" } EQ_Contact(in1 := "KORAK", in2 := 2)
      Contact( "A4+" )
      S_Coil( "A5+_scada" )
      { S7_Templates := "DestType := UInt" } Inc( "KORAK" )
   END_RUNG
   // the same network as SCL:
   IF ("KORAK" = 2) AND "A4+" THEN
       "A5+_scada" := TRUE;
       "KORAK" := "KORAK" + 1;
   END_IF;
END_REGION

REGION Network 6: PC-->PLC
   RUNG wire#powerrail
      { S7_Templates := "SrcType := UInt" } EQ_Contact(in1 := "KORAK", in2 := 3)
      Contact( "A5+" )
      S_Coil( "B2+_scada" )
      { S7_Templates := "DestType := UInt" } Inc( "KORAK" )
   END_RUNG
   // the same network as SCL:
   IF ("KORAK" = 3) AND "A5+" THEN
       "B2+_scada" := TRUE;
       "KORAK" := "KORAK" + 1;
   END_IF;
END_REGION

REGION Network 7: MOTOR SET
   RUNG wire#powerrail
      { S7_Templates := "SrcType := UInt" } EQ_Contact(in1 := "KORAK", in2 := 4)
      Contact( "B2+" )
      { S7_GenerateENO := "TRUE" } Move(in := 10000, out1 => "AnOut4_PUMP")
      { S7_Templates := "DestType := UInt" } Inc( "KORAK" )
   END_RUNG
   // the same network as SCL:
   // ENO of a box is taken as its EN; it also drops when the box reports an error
   IF ("KORAK" = 4) AND "B2+" THEN
       "AnOut4_PUMP" := 10000;
       "KORAK" := "KORAK" + 1;
   END_IF;
END_REGION

REGION Network 8: TIMER
   "TIMER_PROG_1".TONR(IN := "KORAK" = 5, R := "KORAK" <> 5, PT := T#4000MS);
   IF "TIMER_PROG_1".Q AND "dis1_out2" THEN "KORAK" := "KORAK" + 1; END_IF;
END_REGION

REGION Network 9
   RUNG wire#powerrail
      { S7_Templates := "SrcType := UInt" } EQ_Contact(in1 := "KORAK", in2 := 5)
      { S7_Templates := "SrcType := Int" } LE_Contact(in1 := "AnOut4_PUMP", in2 := 25000)
      { S7_Templates := "DestType := Int" } Inc( "AnOut4_PUMP" )
   END_RUNG
   // the same network as SCL:
   IF ("KORAK" = 5) AND ("AnOut4_PUMP" <= 25000) THEN "AnOut4_PUMP" := "AnOut4_PUMP" + 1; END_IF;
END_REGION

REGION Network 10: MOTOR RESET
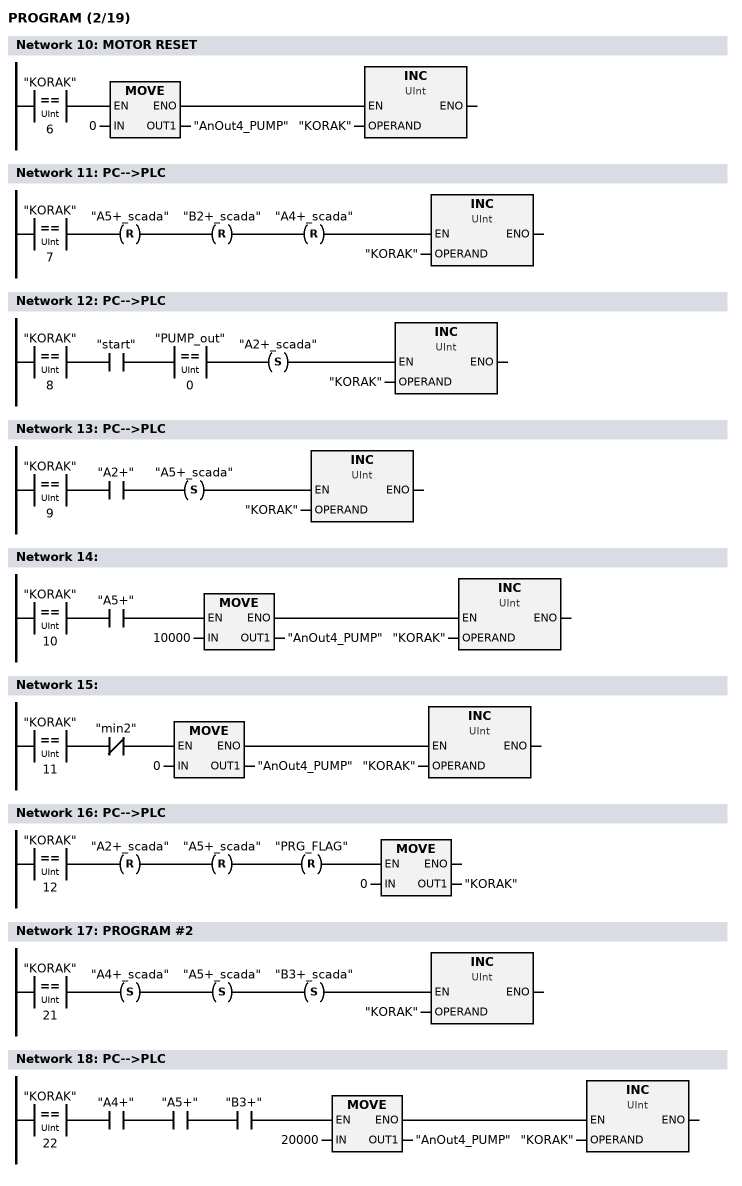
   RUNG wire#powerrail
      { S7_Templates := "SrcType := UInt" } EQ_Contact(in1 := "KORAK", in2 := 6)
      { S7_GenerateENO := "TRUE" } Move(in := 0, out1 => "AnOut4_PUMP")
      { S7_Templates := "DestType := UInt" } Inc( "KORAK" )
   END_RUNG
   // the same network as SCL:
   // ENO of a box is taken as its EN; it also drops when the box reports an error
   IF "KORAK" = 6 THEN
       "AnOut4_PUMP" := 0;
       "KORAK" := "KORAK" + 1;
   END_IF;
END_REGION

REGION Network 11: PC-->PLC
   RUNG wire#powerrail
      { S7_Templates := "SrcType := UInt" } EQ_Contact(in1 := "KORAK", in2 := 7)
      R_Coil( "A5+_scada" )
      R_Coil( "B2+_scada" )
      R_Coil( "A4+_scada" )
      { S7_Templates := "DestType := UInt" } Inc( "KORAK" )
   END_RUNG
   // the same network as SCL:
   IF "KORAK" = 7 THEN
       "A5+_scada" := FALSE;
       "B2+_scada" := FALSE;
       "A4+_scada" := FALSE;
       "KORAK" := "KORAK" + 1;
   END_IF;
END_REGION

REGION Network 12: PC-->PLC
   RUNG wire#powerrail
      { S7_Templates := "SrcType := UInt" } EQ_Contact(in1 := "KORAK", in2 := 8)
      Contact( "start" )
      { S7_Templates := "SrcType := UInt" } EQ_Contact(in1 := "PUMP_out", in2 := 0)
      S_Coil( "A2+_scada" )
      { S7_Templates := "DestType := UInt" } Inc( "KORAK" )
   END_RUNG
   // the same network as SCL:
   IF ("KORAK" = 8) AND "start" AND ("PUMP_out" = 0) THEN
       "A2+_scada" := TRUE;
       "KORAK" := "KORAK" + 1;
   END_IF;
END_REGION

REGION Network 13: PC-->PLC
   RUNG wire#powerrail
      { S7_Templates := "SrcType := UInt" } EQ_Contact(in1 := "KORAK", in2 := 9)
      Contact( "A2+" )
      S_Coil( "A5+_scada" )
      { S7_Templates := "DestType := UInt" } Inc( "KORAK" )
   END_RUNG
   // the same network as SCL:
   IF ("KORAK" = 9) AND "A2+" THEN
       "A5+_scada" := TRUE;
       "KORAK" := "KORAK" + 1;
   END_IF;
END_REGION

REGION Network 14
   RUNG wire#powerrail
      { S7_Templates := "SrcType := UInt" } EQ_Contact(in1 := "KORAK", in2 := 10)
      Contact( "A5+" )
      { S7_GenerateENO := "TRUE" } Move(in := 10000, out1 => "AnOut4_PUMP")
      { S7_Templates := "DestType := UInt" } Inc( "KORAK" )
   END_RUNG
   // the same network as SCL:
   // ENO of a box is taken as its EN; it also drops when the box reports an error
   IF ("KORAK" = 10) AND "A5+" THEN
       "AnOut4_PUMP" := 10000;
       "KORAK" := "KORAK" + 1;
   END_IF;
END_REGION

REGION Network 15
   RUNG wire#powerrail
      { S7_Templates := "SrcType := UInt" } EQ_Contact(in1 := "KORAK", in2 := 11)
      I_Contact( "min2" )
      { S7_GenerateENO := "TRUE" } Move(in := 0, out1 => "AnOut4_PUMP")
      { S7_Templates := "DestType := UInt" } Inc( "KORAK" )
   END_RUNG
   // the same network as SCL:
   // ENO of a box is taken as its EN; it also drops when the box reports an error
   IF ("KORAK" = 11) AND NOT "min2" THEN
       "AnOut4_PUMP" := 0;
       "KORAK" := "KORAK" + 1;
   END_IF;
END_REGION

REGION Network 16: PC-->PLC
   RUNG wire#powerrail
      { S7_Templates := "SrcType := UInt" } EQ_Contact(in1 := "KORAK", in2 := 12)
      R_Coil( "A2+_scada" )
      R_Coil( "A5+_scada" )
      R_Coil( "PRG_FLAG" )
      Move(in := 0, out1 => "KORAK")
   END_RUNG
   // the same network as SCL:
   IF "KORAK" = 12 THEN
       "A2+_scada" := FALSE;
       "A5+_scada" := FALSE;
       "PRG_FLAG" := FALSE;
       "KORAK" := 0;
   END_IF;
END_REGION

REGION Network 17: PROGRAM #2
   RUNG wire#powerrail
      { S7_Templates := "SrcType := UInt" } EQ_Contact(in1 := "KORAK", in2 := 21)
      S_Coil( "A4+_scada" )
      S_Coil( "A5+_scada" )
      S_Coil( "B3+_scada" )
      { S7_Templates := "DestType := UInt" } Inc( "KORAK" )
   END_RUNG
   // the same network as SCL:
   IF "KORAK" = 21 THEN
       "A4+_scada" := TRUE;
       "A5+_scada" := TRUE;
       "B3+_scada" := TRUE;
       "KORAK" := "KORAK" + 1;
   END_IF;
END_REGION

REGION Network 18: PC-->PLC
   RUNG wire#powerrail
      { S7_Templates := "SrcType := UInt" } EQ_Contact(in1 := "KORAK", in2 := 22)
      Contact( "A4+" )
      Contact( "A5+" )
      Contact( "B3+" )
      { S7_GenerateENO := "TRUE" } Move(in := 20000, out1 => "AnOut4_PUMP")
      { S7_Templates := "DestType := UInt" } Inc( "KORAK" )
   END_RUNG
   // the same network as SCL:
   // ENO of a box is taken as its EN; it also drops when the box reports an error
   IF ("KORAK" = 22) AND "A4+" AND "A5+" AND "B3+" THEN
       "AnOut4_PUMP" := 20000;
       "KORAK" := "KORAK" + 1;
   END_IF;
END_REGION

REGION Network 19: PC-->PLC
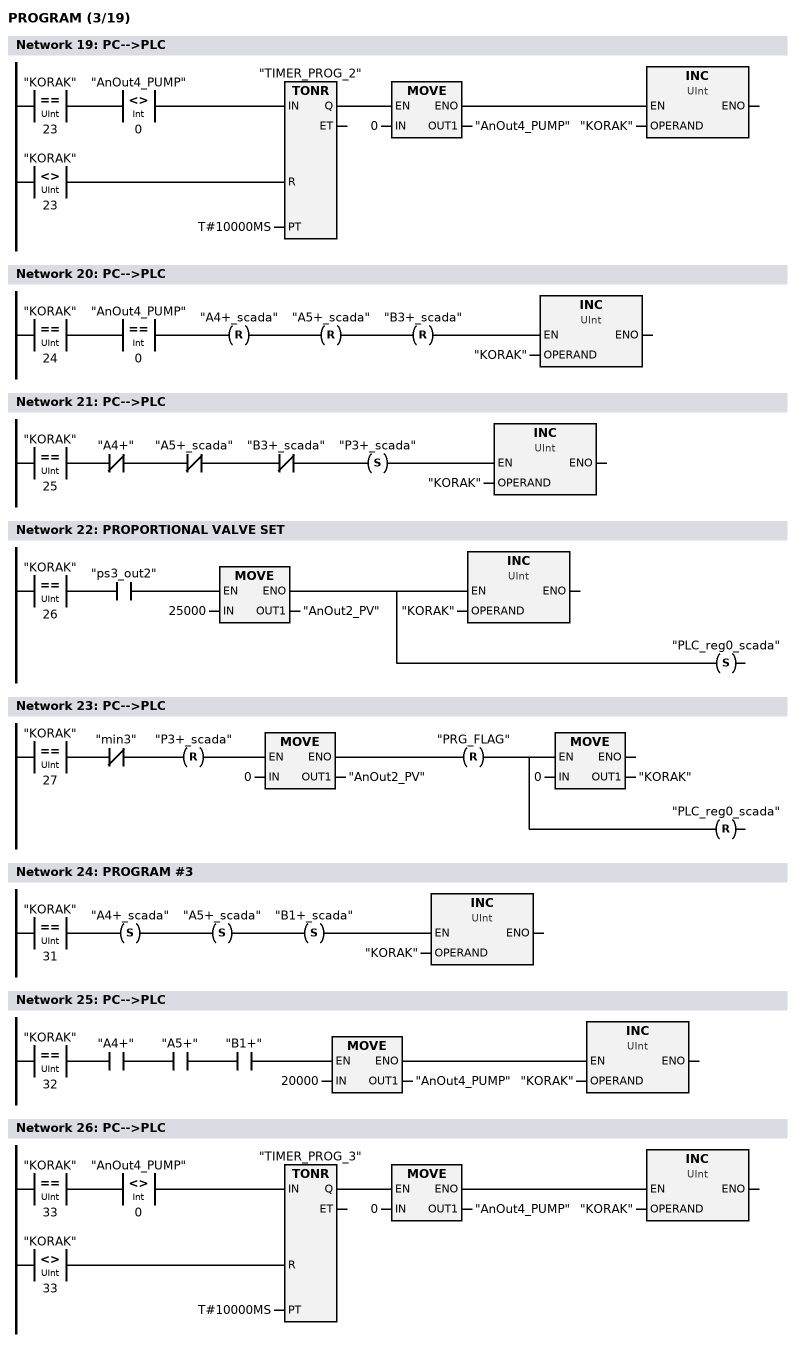
   // ENO of a box is taken as its EN; it also drops when the box reports an error
   "TIMER_PROG_2".TONR(IN := ("KORAK" = 23) AND ("AnOut4_PUMP" <> 0), R := "KORAK" <> 23, PT := T#10000MS);
   IF "TIMER_PROG_2".Q THEN
       "AnOut4_PUMP" := 0;
       "KORAK" := "KORAK" + 1;
   END_IF;
END_REGION

REGION Network 20: PC-->PLC
   RUNG wire#powerrail
      { S7_Templates := "SrcType := UInt" } EQ_Contact(in1 := "KORAK", in2 := 24)
      { S7_Templates := "SrcType := Int" } EQ_Contact(in1 := "AnOut4_PUMP", in2 := 0)
      R_Coil( "A4+_scada" )
      R_Coil( "A5+_scada" )
      R_Coil( "B3+_scada" )
      { S7_Templates := "DestType := UInt" } Inc( "KORAK" )
   END_RUNG
   // the same network as SCL:
   IF ("KORAK" = 24) AND ("AnOut4_PUMP" = 0) THEN
       "A4+_scada" := FALSE;
       "A5+_scada" := FALSE;
       "B3+_scada" := FALSE;
       "KORAK" := "KORAK" + 1;
   END_IF;
END_REGION

REGION Network 21: PC-->PLC
   RUNG wire#powerrail
      { S7_Templates := "SrcType := UInt" } EQ_Contact(in1 := "KORAK", in2 := 25)
      I_Contact( "A4+" )
      I_Contact( "A5+_scada" )
      I_Contact( "B3+_scada" )
      S_Coil( "P3+_scada" )
      { S7_Templates := "DestType := UInt" } Inc( "KORAK" )
   END_RUNG
   // the same network as SCL:
   IF ("KORAK" = 25) AND NOT "A4+" AND NOT "A5+_scada" AND NOT "B3+_scada" THEN
       "P3+_scada" := TRUE;
       "KORAK" := "KORAK" + 1;
   END_IF;
END_REGION

REGION Network 22: PROPORTIONAL VALVE SET
   RUNG wire#powerrail
      { S7_Templates := "SrcType := UInt" } EQ_Contact(in1 := "KORAK", in2 := 26)
      Contact( "ps3_out2" )
      { S7_GenerateENO := "TRUE" } Move(in := 25000, out1 => "AnOut2_PV")
      wire#w1
      { S7_Templates := "DestType := UInt" } Inc( "KORAK" )
   END_RUNG
   RUNG wire#w1
      S_Coil( "PLC_reg0_scada" )
   END_RUNG
   // the same network as SCL:
   // ENO of a box is taken as its EN; it also drops when the box reports an error
   IF ("KORAK" = 26) AND "ps3_out2" THEN "AnOut2_PV" := 25000; END_IF;
   #_w1 := ("KORAK" = 26) AND "ps3_out2";
   IF #_w1 THEN
       "KORAK" := "KORAK" + 1;
       "PLC_reg0_scada" := TRUE;
   END_IF;
END_REGION

REGION Network 23: PC-->PLC
   RUNG wire#powerrail
      { S7_Templates := "SrcType := UInt" } EQ_Contact(in1 := "KORAK", in2 := 27)
      I_Contact( "min3" )
      R_Coil( "P3+_scada" )
      { S7_GenerateENO := "TRUE" } Move(in := 0, out1 => "AnOut2_PV")
      R_Coil( "PRG_FLAG" )
      wire#w1
      { S7_GenerateENO := "TRUE" } Move(in := 0, out1 => "KORAK")
   END_RUNG
   RUNG wire#w1
      R_Coil( "PLC_reg0_scada" )
   END_RUNG
   // the same network as SCL:
   // ENO of a box is taken as its EN; it also drops when the box reports an error
   IF ("KORAK" = 27) AND NOT "min3" THEN
       "P3+_scada" := FALSE;
       "AnOut2_PV" := 0;
       "PRG_FLAG" := FALSE;
   END_IF;
   #_w1 := ("KORAK" = 27) AND NOT "min3";
   IF #_w1 THEN
       "KORAK" := 0;
       "PLC_reg0_scada" := FALSE;
   END_IF;
END_REGION

REGION Network 24: PROGRAM #3
   RUNG wire#powerrail
      { S7_Templates := "SrcType := UInt" } EQ_Contact(in1 := "KORAK", in2 := 31)
      S_Coil( "A4+_scada" )
      S_Coil( "A5+_scada" )
      S_Coil( "B1+_scada" )
      { S7_Templates := "DestType := UInt" } Inc( "KORAK" )
   END_RUNG
   // the same network as SCL:
   IF "KORAK" = 31 THEN
       "A4+_scada" := TRUE;
       "A5+_scada" := TRUE;
       "B1+_scada" := TRUE;
       "KORAK" := "KORAK" + 1;
   END_IF;
END_REGION

REGION Network 25: PC-->PLC
   RUNG wire#powerrail
      { S7_Templates := "SrcType := UInt" } EQ_Contact(in1 := "KORAK", in2 := 32)
      Contact( "A4+" )
      Contact( "A5+" )
      Contact( "B1+" )
      { S7_GenerateENO := "TRUE" } Move(in := 20000, out1 => "AnOut4_PUMP")
      { S7_Templates := "DestType := UInt" } Inc( "KORAK" )
   END_RUNG
   // the same network as SCL:
   // ENO of a box is taken as its EN; it also drops when the box reports an error
   IF ("KORAK" = 32) AND "A4+" AND "A5+" AND "B1+" THEN
       "AnOut4_PUMP" := 20000;
       "KORAK" := "KORAK" + 1;
   END_IF;
END_REGION

REGION Network 26: PC-->PLC
   // ENO of a box is taken as its EN; it also drops when the box reports an error
   "TIMER_PROG_3".TONR(IN := ("KORAK" = 33) AND ("AnOut4_PUMP" <> 0), R := "KORAK" <> 33, PT := T#10000MS);
   IF "TIMER_PROG_3".Q THEN
       "AnOut4_PUMP" := 0;
       "KORAK" := "KORAK" + 1;
   END_IF;
END_REGION

REGION Network 27: PC-->PLC
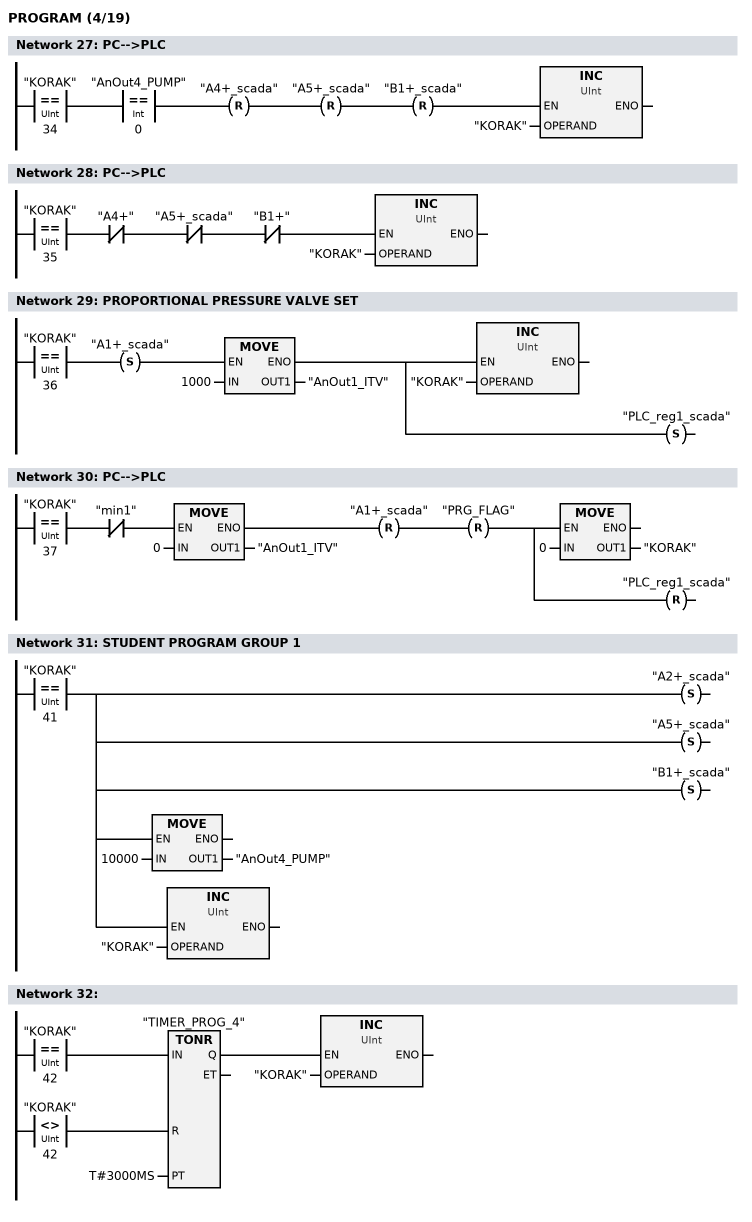
   RUNG wire#powerrail
      { S7_Templates := "SrcType := UInt" } EQ_Contact(in1 := "KORAK", in2 := 34)
      { S7_Templates := "SrcType := Int" } EQ_Contact(in1 := "AnOut4_PUMP", in2 := 0)
      R_Coil( "A4+_scada" )
      R_Coil( "A5+_scada" )
      R_Coil( "B1+_scada" )
      { S7_Templates := "DestType := UInt" } Inc( "KORAK" )
   END_RUNG
   // the same network as SCL:
   IF ("KORAK" = 34) AND ("AnOut4_PUMP" = 0) THEN
       "A4+_scada" := FALSE;
       "A5+_scada" := FALSE;
       "B1+_scada" := FALSE;
       "KORAK" := "KORAK" + 1;
   END_IF;
END_REGION

REGION Network 28: PC-->PLC
   RUNG wire#powerrail
      { S7_Templates := "SrcType := UInt" } EQ_Contact(in1 := "KORAK", in2 := 35)
      I_Contact( "A4+" )
      I_Contact( "A5+_scada" )
      I_Contact( "B1+" )
      { S7_Templates := "DestType := UInt" } Inc( "KORAK" )
   END_RUNG
   // the same network as SCL:
   IF ("KORAK" = 35) AND NOT "A4+" AND NOT "A5+_scada" AND NOT "B1+" THEN "KORAK" := "KORAK" + 1; END_IF;
END_REGION

REGION Network 29: PROPORTIONAL PRESSURE VALVE SET
   RUNG wire#powerrail
      { S7_Templates := "SrcType := UInt" } EQ_Contact(in1 := "KORAK", in2 := 36)
      S_Coil( "A1+_scada" )
      { S7_GenerateENO := "TRUE" } Move(in := 1000, out1 => "AnOut1_ITV")
      wire#w1
      { S7_Templates := "DestType := UInt" } Inc( "KORAK" )
   END_RUNG
   RUNG wire#w1
      S_Coil( "PLC_reg1_scada" )
   END_RUNG
   // the same network as SCL:
   // ENO of a box is taken as its EN; it also drops when the box reports an error
   IF "KORAK" = 36 THEN
       "A1+_scada" := TRUE;
       "AnOut1_ITV" := 1000;
   END_IF;
   #_w1 := "KORAK" = 36;
   IF #_w1 THEN
       "KORAK" := "KORAK" + 1;
       "PLC_reg1_scada" := TRUE;
   END_IF;
END_REGION

REGION Network 30: PC-->PLC
   RUNG wire#powerrail
      { S7_Templates := "SrcType := UInt" } EQ_Contact(in1 := "KORAK", in2 := 37)
      I_Contact( "min1" )
      { S7_GenerateENO := "TRUE" } Move(in := 0, out1 => "AnOut1_ITV")
      R_Coil( "A1+_scada" )
      R_Coil( "PRG_FLAG" )
      wire#w1
      { S7_GenerateENO := "TRUE" } Move(in := 0, out1 => "KORAK")
   END_RUNG
   RUNG wire#w1
      R_Coil( "PLC_reg1_scada" )
   END_RUNG
   // the same network as SCL:
   // ENO of a box is taken as its EN; it also drops when the box reports an error
   IF ("KORAK" = 37) AND NOT "min1" THEN
       "AnOut1_ITV" := 0;
       "A1+_scada" := FALSE;
       "PRG_FLAG" := FALSE;
   END_IF;
   #_w1 := ("KORAK" = 37) AND NOT "min1";
   IF #_w1 THEN
       "KORAK" := 0;
       "PLC_reg1_scada" := FALSE;
   END_IF;
END_REGION

REGION Network 31: STUDENT PROGRAM GROUP 1
   RUNG wire#powerrail
      { S7_Templates := "SrcType := UInt" } EQ_Contact(in1 := "KORAK", in2 := 41)
      wire#w1
      S_Coil( "A2+_scada" )
   END_RUNG
   RUNG wire#w1
      S_Coil( "A5+_scada" )
   END_RUNG
   RUNG wire#w1
      S_Coil( "B1+_scada" )
   END_RUNG
   RUNG wire#w1
      { S7_GenerateENO := "TRUE" } Move(in := 10000, out1 => "AnOut4_PUMP")
   END_RUNG
   RUNG wire#w1
      { S7_Templates := "DestType := UInt" } Inc( "KORAK" )
   END_RUNG
   // the same network as SCL:
   IF "KORAK" = 41 THEN
       "A2+_scada" := TRUE;
       "A5+_scada" := TRUE;
       "B1+_scada" := TRUE;
       "AnOut4_PUMP" := 10000;
       "KORAK" := "KORAK" + 1;
   END_IF;
END_REGION

REGION Network 32
   "TIMER_PROG_4".TONR(IN := "KORAK" = 42, R := "KORAK" <> 42, PT := T#3000MS);
   IF "TIMER_PROG_4".Q THEN "KORAK" := "KORAK" + 1; END_IF;
END_REGION

REGION Network 33: PC-->PLC
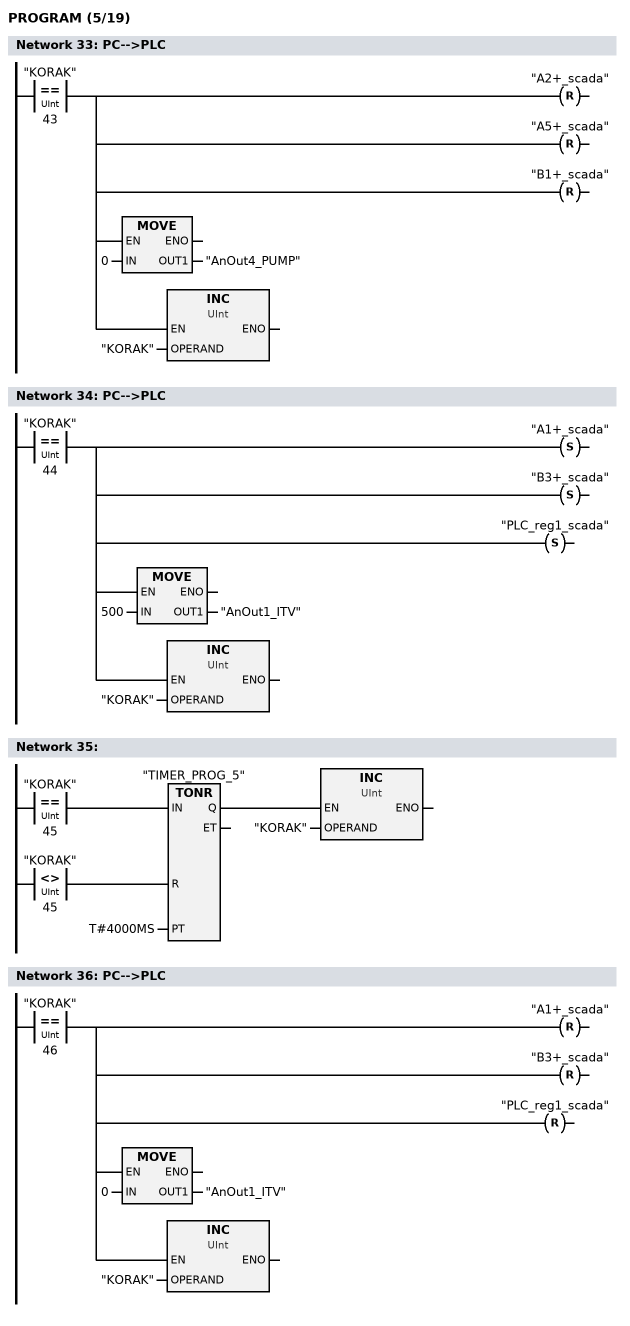
   RUNG wire#powerrail
      { S7_Templates := "SrcType := UInt" } EQ_Contact(in1 := "KORAK", in2 := 43)
      wire#w1
      R_Coil( "A2+_scada" )
   END_RUNG
   RUNG wire#w1
      R_Coil( "A5+_scada" )
   END_RUNG
   RUNG wire#w1
      R_Coil( "B1+_scada" )
   END_RUNG
   RUNG wire#w1
      { S7_GenerateENO := "TRUE" } Move(in := 0, out1 => "AnOut4_PUMP")
   END_RUNG
   RUNG wire#w1
      { S7_Templates := "DestType := UInt" } Inc( "KORAK" )
   END_RUNG
   // the same network as SCL:
   IF "KORAK" = 43 THEN
       "A2+_scada" := FALSE;
       "A5+_scada" := FALSE;
       "B1+_scada" := FALSE;
       "AnOut4_PUMP" := 0;
       "KORAK" := "KORAK" + 1;
   END_IF;
END_REGION

REGION Network 34: PC-->PLC
   RUNG wire#powerrail
      { S7_Templates := "SrcType := UInt" } EQ_Contact(in1 := "KORAK", in2 := 44)
      wire#w1
      S_Coil( "A1+_scada" )
   END_RUNG
   RUNG wire#w1
      S_Coil( "B3+_scada" )
   END_RUNG
   RUNG wire#w1
      S_Coil( "PLC_reg1_scada" )
   END_RUNG
   RUNG wire#w1
      { S7_GenerateENO := "TRUE" } Move(in := 500, out1 => "AnOut1_ITV")
   END_RUNG
   RUNG wire#w1
      { S7_Templates := "DestType := UInt" } Inc( "KORAK" )
   END_RUNG
   // the same network as SCL:
   IF "KORAK" = 44 THEN
       "A1+_scada" := TRUE;
       "B3+_scada" := TRUE;
       "PLC_reg1_scada" := TRUE;
       "AnOut1_ITV" := 500;
       "KORAK" := "KORAK" + 1;
   END_IF;
END_REGION

REGION Network 35
   "TIMER_PROG_5".TONR(IN := "KORAK" = 45, R := "KORAK" <> 45, PT := T#4000MS);
   IF "TIMER_PROG_5".Q THEN "KORAK" := "KORAK" + 1; END_IF;
END_REGION

REGION Network 36: PC-->PLC
   RUNG wire#powerrail
      { S7_Templates := "SrcType := UInt" } EQ_Contact(in1 := "KORAK", in2 := 46)
      wire#w1
      R_Coil( "A1+_scada" )
   END_RUNG
   RUNG wire#w1
      R_Coil( "B3+_scada" )
   END_RUNG
   RUNG wire#w1
      R_Coil( "PLC_reg1_scada" )
   END_RUNG
   RUNG wire#w1
      { S7_GenerateENO := "TRUE" } Move(in := 0, out1 => "AnOut1_ITV")
   END_RUNG
   RUNG wire#w1
      { S7_Templates := "DestType := UInt" } Inc( "KORAK" )
   END_RUNG
   // the same network as SCL:
   IF "KORAK" = 46 THEN
       "A1+_scada" := FALSE;
       "B3+_scada" := FALSE;
       "PLC_reg1_scada" := FALSE;
       "AnOut1_ITV" := 0;
       "KORAK" := "KORAK" + 1;
   END_IF;
END_REGION

REGION Network 37: PC-->PLC
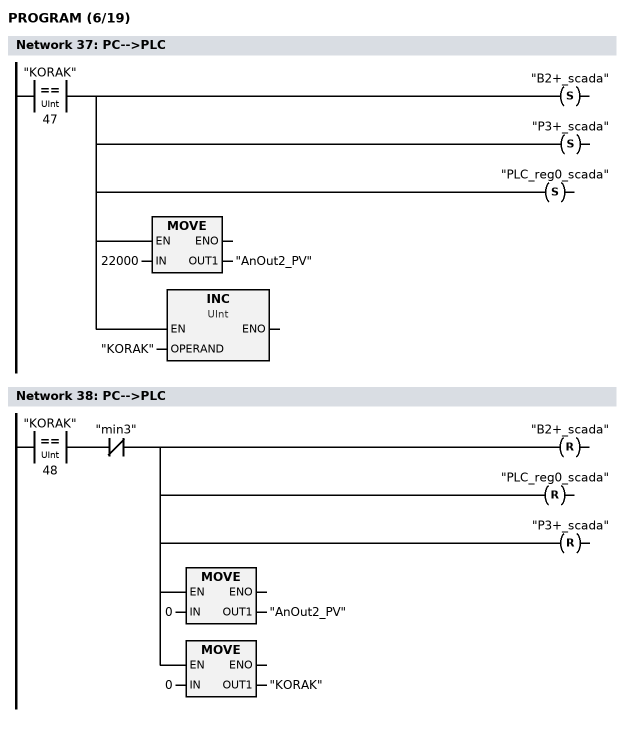
   RUNG wire#powerrail
      { S7_Templates := "SrcType := UInt" } EQ_Contact(in1 := "KORAK", in2 := 47)
      wire#w1
      S_Coil( "B2+_scada" )
   END_RUNG
   RUNG wire#w1
      S_Coil( "P3+_scada" )
   END_RUNG
   RUNG wire#w1
      S_Coil( "PLC_reg0_scada" )
   END_RUNG
   RUNG wire#w1
      { S7_GenerateENO := "TRUE" } Move(in := 22000, out1 => "AnOut2_PV")
   END_RUNG
   RUNG wire#w1
      { S7_Templates := "DestType := UInt" } Inc( "KORAK" )
   END_RUNG
   // the same network as SCL:
   IF "KORAK" = 47 THEN
       "B2+_scada" := TRUE;
       "P3+_scada" := TRUE;
       "PLC_reg0_scada" := TRUE;
       "AnOut2_PV" := 22000;
       "KORAK" := "KORAK" + 1;
   END_IF;
END_REGION

REGION Network 38: PC-->PLC
   RUNG wire#powerrail
      { S7_Templates := "SrcType := UInt" } EQ_Contact(in1 := "KORAK", in2 := 48)
      I_Contact( "min3" )
      wire#w1
      R_Coil( "B2+_scada" )
   END_RUNG
   RUNG wire#w1
      R_Coil( "PLC_reg0_scada" )
   END_RUNG
   RUNG wire#w1
      R_Coil( "P3+_scada" )
   END_RUNG
   RUNG wire#w1
      { S7_GenerateENO := "TRUE" } Move(in := 0, out1 => "AnOut2_PV")
   END_RUNG
   RUNG wire#w1
      { S7_GenerateENO := "TRUE" } Move(in := 0, out1 => "KORAK")
   END_RUNG
   // the same network as SCL:
   IF ("KORAK" = 48) AND NOT "min3" THEN
       "B2+_scada" := FALSE;
       "PLC_reg0_scada" := FALSE;
       "P3+_scada" := FALSE;
       "AnOut2_PV" := 0;
       "KORAK" := 0;
   END_IF;
END_REGION

REGION Network 39: STUDENT PROGRAM GROUP 2
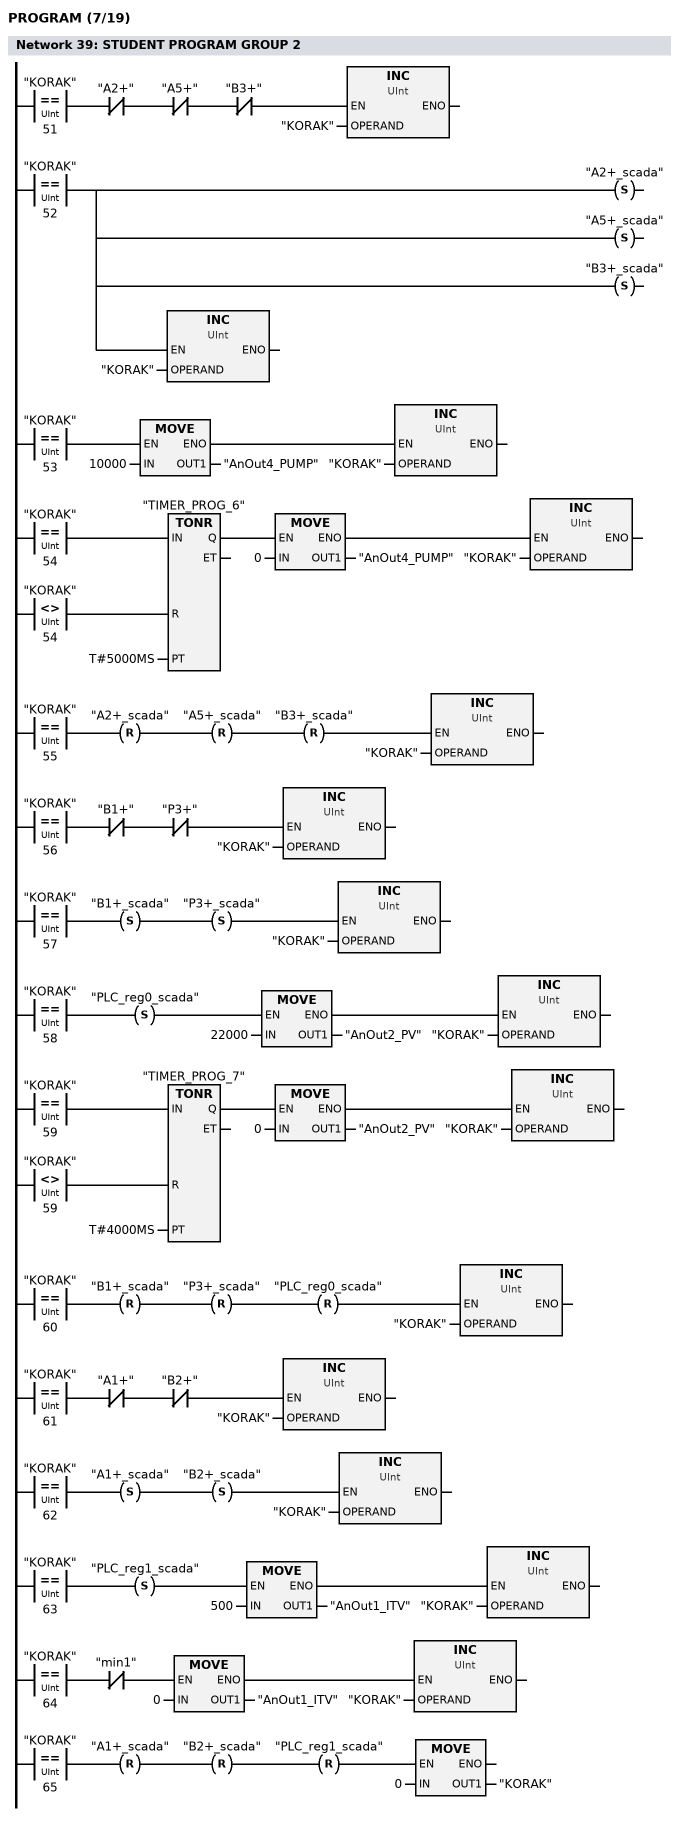
   // ENO of a box is taken as its EN; it also drops when the box reports an error
   IF ("KORAK" = 51) AND NOT "A2+" AND NOT "A5+" AND NOT "B3+" THEN "KORAK" := "KORAK" + 1; END_IF;
   IF "KORAK" = 52 THEN
       "A2+_scada" := TRUE;
       "A5+_scada" := TRUE;
       "B3+_scada" := TRUE;
       "KORAK" := "KORAK" + 1;
   END_IF;
   IF "KORAK" = 53 THEN
       "AnOut4_PUMP" := 10000;
       "KORAK" := "KORAK" + 1;
   END_IF;
   "TIMER_PROG_6".TONR(IN := "KORAK" = 54, R := "KORAK" <> 54, PT := T#5000MS);
   IF "TIMER_PROG_6".Q THEN
       "AnOut4_PUMP" := 0;
       "KORAK" := "KORAK" + 1;
   END_IF;
   IF "KORAK" = 55 THEN
       "A2+_scada" := FALSE;
       "A5+_scada" := FALSE;
       "B3+_scada" := FALSE;
       "KORAK" := "KORAK" + 1;
   END_IF;
   IF ("KORAK" = 56) AND NOT "B1+" AND NOT "P3+" THEN "KORAK" := "KORAK" + 1; END_IF;
   IF "KORAK" = 57 THEN
       "B1+_scada" := TRUE;
       "P3+_scada" := TRUE;
       "KORAK" := "KORAK" + 1;
   END_IF;
   IF "KORAK" = 58 THEN
       "PLC_reg0_scada" := TRUE;
       "AnOut2_PV" := 22000;
       "KORAK" := "KORAK" + 1;
   END_IF;
   "TIMER_PROG_7".TONR(IN := "KORAK" = 59, R := "KORAK" <> 59, PT := T#4000MS);
   IF "TIMER_PROG_7".Q THEN
       "AnOut2_PV" := 0;
       "KORAK" := "KORAK" + 1;
   END_IF;
   IF "KORAK" = 60 THEN
       "B1+_scada" := FALSE;
       "P3+_scada" := FALSE;
       "PLC_reg0_scada" := FALSE;
       "KORAK" := "KORAK" + 1;
   END_IF;
   IF ("KORAK" = 61) AND NOT "A1+" AND NOT "B2+" THEN "KORAK" := "KORAK" + 1; END_IF;
   IF "KORAK" = 62 THEN
       "A1+_scada" := TRUE;
       "B2+_scada" := TRUE;
       "KORAK" := "KORAK" + 1;
   END_IF;
   IF "KORAK" = 63 THEN
       "PLC_reg1_scada" := TRUE;
       "AnOut1_ITV" := 500;
       "KORAK" := "KORAK" + 1;
   END_IF;
   IF ("KORAK" = 64) AND NOT "min1" THEN
       "AnOut1_ITV" := 0;
       "KORAK" := "KORAK" + 1;
   END_IF;
   IF "KORAK" = 65 THEN
       "A1+_scada" := FALSE;
       "B2+_scada" := FALSE;
       "PLC_reg1_scada" := FALSE;
       "KORAK" := 0;
   END_IF;
END_REGION

REGION Network 40: STUDENT PROGRAM GROUP 21
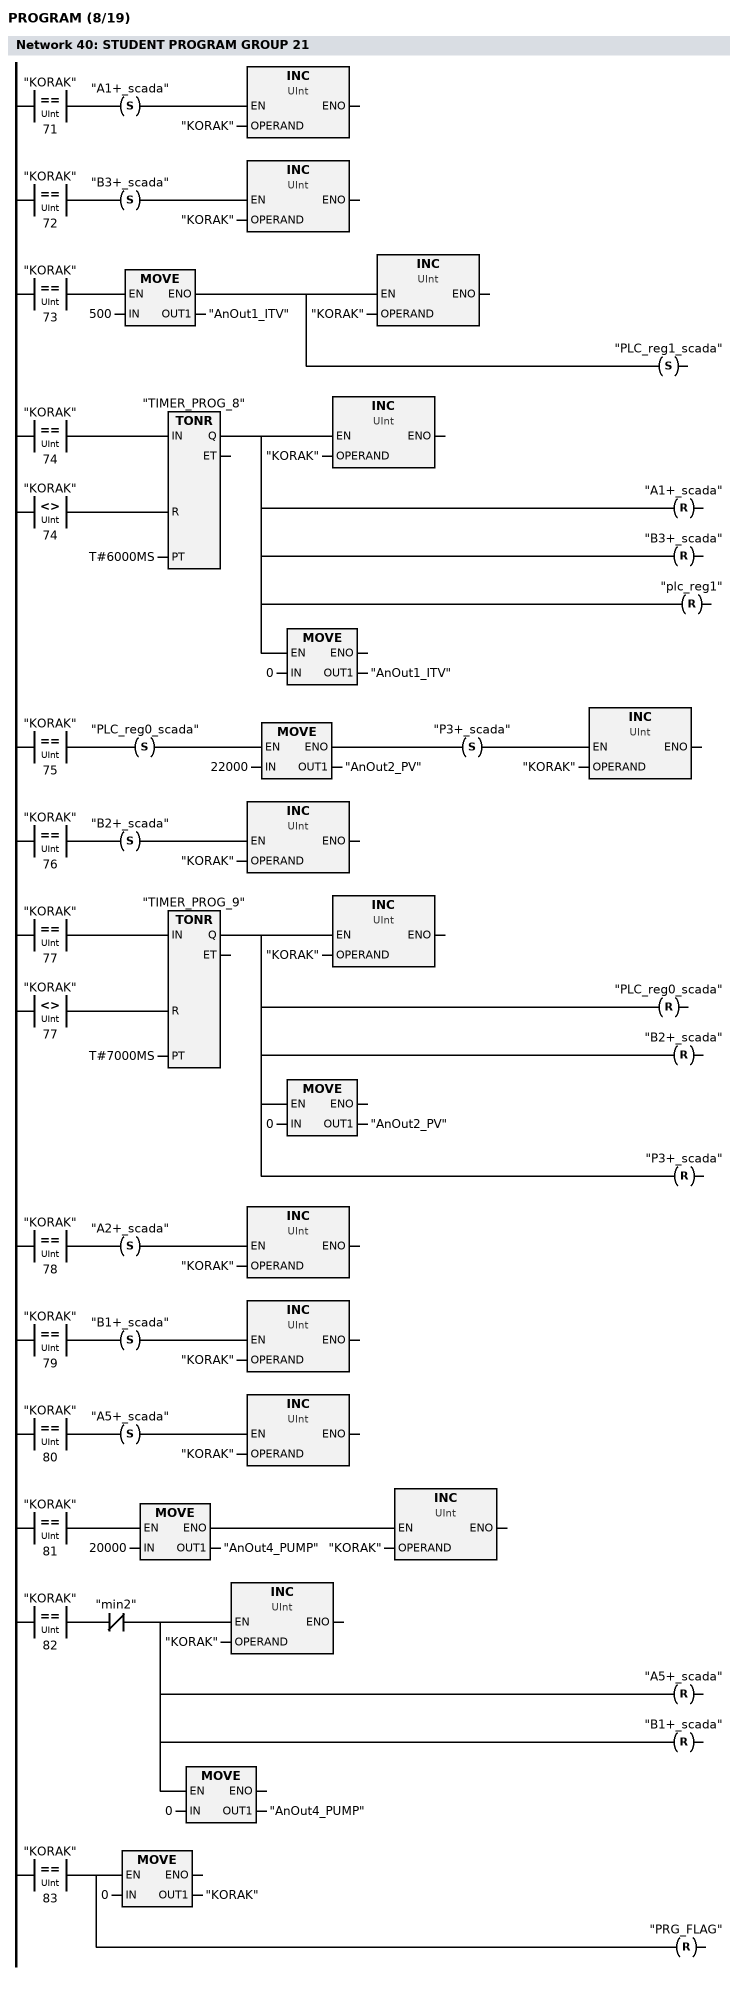
   IF "KORAK" = 71 THEN
       "A1+_scada" := TRUE;
       "KORAK" := "KORAK" + 1;
   END_IF;
   IF "KORAK" = 72 THEN
       "B3+_scada" := TRUE;
       "KORAK" := "KORAK" + 1;
   END_IF;
   IF "KORAK" = 73 THEN "AnOut1_ITV" := 500; END_IF;
   #_w1 := "KORAK" = 73;
   IF #_w1 THEN
       "KORAK" := "KORAK" + 1;
       "PLC_reg1_scada" := TRUE;
   END_IF;
   "TIMER_PROG_8".TONR(IN := "KORAK" = 74, R := "KORAK" <> 74, PT := T#6000MS);
   IF "TIMER_PROG_8".Q THEN
       "KORAK" := "KORAK" + 1;
       "A1+_scada" := FALSE;
       "B3+_scada" := FALSE;
       "plc_reg1" := FALSE;
       "AnOut1_ITV" := 0;
   END_IF;
   IF "KORAK" = 75 THEN
       "PLC_reg0_scada" := TRUE;
       "AnOut2_PV" := 22000;
       "P3+_scada" := TRUE;
       "KORAK" := "KORAK" + 1;
   END_IF;
   IF "KORAK" = 76 THEN
       "B2+_scada" := TRUE;
       "KORAK" := "KORAK" + 1;
   END_IF;
   "TIMER_PROG_9".TONR(IN := "KORAK" = 77, R := "KORAK" <> 77, PT := T#7000MS);
   IF "TIMER_PROG_9".Q THEN
       "KORAK" := "KORAK" + 1;
       "PLC_reg0_scada" := FALSE;
       "B2+_scada" := FALSE;
       "AnOut2_PV" := 0;
       "P3+_scada" := FALSE;
   END_IF;
   IF "KORAK" = 78 THEN
       "A2+_scada" := TRUE;
       "KORAK" := "KORAK" + 1;
   END_IF;
   IF "KORAK" = 79 THEN
       "B1+_scada" := TRUE;
       "KORAK" := "KORAK" + 1;
   END_IF;
   IF "KORAK" = 80 THEN
       "A5+_scada" := TRUE;
       "KORAK" := "KORAK" + 1;
   END_IF;
   IF "KORAK" = 81 THEN
       "AnOut4_PUMP" := 20000;
       "KORAK" := "KORAK" + 1;
   END_IF;
   #_w2 := ("KORAK" = 82) AND NOT "min2";
   IF #_w2 THEN
       "KORAK" := "KORAK" + 1;
       "A5+_scada" := FALSE;
       "B1+_scada" := FALSE;
       "AnOut4_PUMP" := 0;
   END_IF;
   #_w3 := "KORAK" = 83;
   IF #_w3 THEN
       "KORAK" := 0;
       "PRG_FLAG" := FALSE;
   END_IF;
END_REGION

REGION Network 41: PC-->PLC
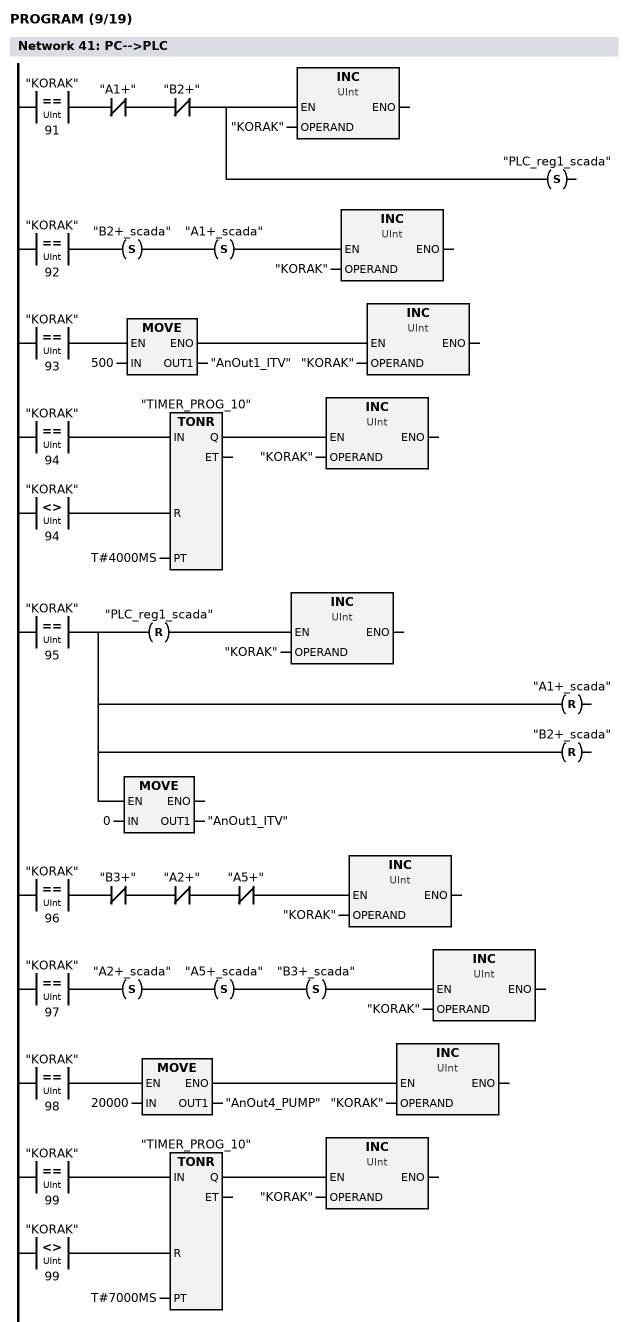
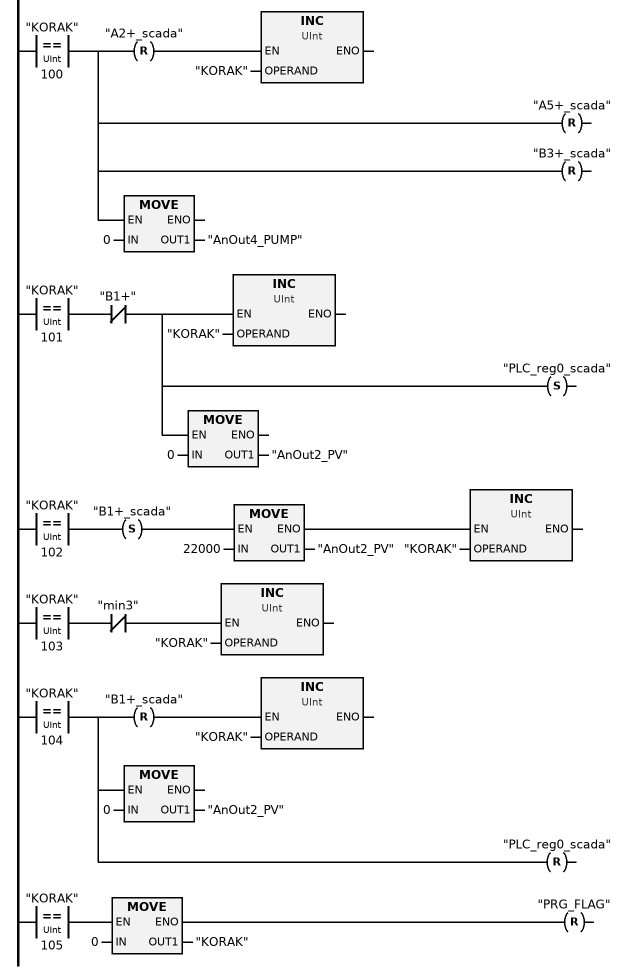
   #_w1 := ("KORAK" = 91) AND NOT "A1+" AND NOT "B2+";
   IF #_w1 THEN
       "KORAK" := "KORAK" + 1;
       "PLC_reg1_scada" := TRUE;
   END_IF;
   IF "KORAK" = 92 THEN
       "B2+_scada" := TRUE;
       "A1+_scada" := TRUE;
       "KORAK" := "KORAK" + 1;
   END_IF;
   IF "KORAK" = 93 THEN
       "AnOut1_ITV" := 500;
       "KORAK" := "KORAK" + 1;
   END_IF;
   "TIMER_PROG_10".TONR(IN := "KORAK" = 94, R := "KORAK" <> 94, PT := T#4000MS);
   IF "TIMER_PROG_10".Q THEN "KORAK" := "KORAK" + 1; END_IF;
   IF "KORAK" = 95 THEN "PLC_reg1_scada" := FALSE; END_IF;
   #_w2 := "KORAK" = 95;
   IF #_w2 THEN
       "KORAK" := "KORAK" + 1;
       "A1+_scada" := FALSE;
       "B2+_scada" := FALSE;
       "AnOut1_ITV" := 0;
   END_IF;
   IF ("KORAK" = 96) AND NOT "B3+" AND NOT "A2+" AND NOT "A5+" THEN "KORAK" := "KORAK" + 1; END_IF;
   IF "KORAK" = 97 THEN
       "A2+_scada" := TRUE;
       "A5+_scada" := TRUE;
       "B3+_scada" := TRUE;
       "KORAK" := "KORAK" + 1;
   END_IF;
   IF "KORAK" = 98 THEN
       "AnOut4_PUMP" := 20000;
       "KORAK" := "KORAK" + 1;
   END_IF;
   "TIMER_PROG_10".TONR(IN := "KORAK" = 99, R := "KORAK" <> 99, PT := T#7000MS);
   IF "TIMER_PROG_10".Q THEN "KORAK" := "KORAK" + 1; END_IF;
   IF "KORAK" = 100 THEN "A2+_scada" := FALSE; END_IF;
   #_w3 := "KORAK" = 100;
   IF #_w3 THEN
       "KORAK" := "KORAK" + 1;
       "A5+_scada" := FALSE;
       "B3+_scada" := FALSE;
       "AnOut4_PUMP" := 0;
   END_IF;
   #_w4 := ("KORAK" = 101) AND NOT "B1+";
   IF #_w4 THEN
       "KORAK" := "KORAK" + 1;
       "PLC_reg0_scada" := TRUE;
       "AnOut2_PV" := 0;
   END_IF;
   IF "KORAK" = 102 THEN
       "B1+_scada" := TRUE;
       "AnOut2_PV" := 22000;
       "KORAK" := "KORAK" + 1;
   END_IF;
   IF ("KORAK" = 103) AND NOT "min3" THEN "KORAK" := "KORAK" + 1; END_IF;
   IF "KORAK" = 104 THEN "B1+_scada" := FALSE; END_IF;
   #_w5 := "KORAK" = 104;
   IF #_w5 THEN
       "KORAK" := "KORAK" + 1;
       "AnOut2_PV" := 0;
       "PLC_reg0_scada" := FALSE;
   END_IF;
   #_w6 := "KORAK" = 105;
   IF #_w6 THEN
       "KORAK" := 0;
       "PRG_FLAG" := FALSE;
   END_IF;
END_REGION

REGION Network 42: PC-->PLC
